									[9].arrDataOut[59]	:=	<0, 8, 8>TIIB(104)^API^Data^io^Outputs^Request Data[29];
									[9].arrDataOut[60]	:=	<0, 8, 0>TIIB(104)^API^Data^io^Outputs^Request Data[30];
									[9].arrDataOut[61]	:=	<0, 8, 8>TIIB(104)^API^Data^io^Outputs^Request Data[30];
									[9].arrDataOut[62]	:=	<0, 8, 0>TIIB(104)^API^Data^io^Outputs^Request Data[31];
									[9].arrDataOut[63]	:=	<0, 8, 8>TIIB(104)^API^Data^io^Outputs^Request Data[31];
									[9].PnIoBoxState 	:=	<0, 16, 0>TIIB(104)^Inputs^PnIoBoxState;
									[10].arrDataIn[0]	:=	<0, 8, 0>TIIB(105)^API^Data^io^Inputs^Response Data[0];
									[10].arrDataIn[1]	:=	<0, 8, 8>TIIB(105)^API^Data^io^Inputs^Response Data[0];
									[10].arrDataIn[2]	:=	<0, 8, 0>TIIB(105)^API^Data^io^Inputs^Response Data[1];
									[10].arrDataIn[3]	:=	<0, 8, 8>TIIB(105)^API^Data^io^Inputs^Response Data[1];
									[10].arrDataIn[4]	:=	<0, 8, 0>TIIB(105)^API^Data^io^Inputs^Response Data[2];
									[10].arrDataIn[5]	:=	<0, 8, 8>TIIB(105)^API^Data^io^Inputs^Response Data[2];
									[10].arrDataIn[6]	:=	<0, 8, 0>TIIB(105)^API^Data^io^Inputs^Response Data[3];
									[10].arrDataIn[7]	:=	<0, 8, 8>TIIB(105)^API^Data^io^Inputs^Response Data[3];
									[10].arrDataIn[8]	:=	<0, 8, 0>TIIB(105)^API^Data^io^Inputs^Response Data[4];
									[10].arrDataIn[9]	:=	<0, 8, 8>TIIB(105)^API^Data^io^Inputs^Response Data[4];
									[10].arrDataIn[10]	:=	<0, 8, 0>TIIB(105)^API^Data^io^Inputs^Response Data[5];
									[10].arrDataIn[11]	:=	<0, 8, 8>TIIB(105)^API^Data^io^Inputs^Response Data[5];
									[10].arrDataIn[12]	:=	<0, 8, 0>TIIB(105)^API^Data^io^Inputs^Response Data[6];
									[10].arrDataIn[13]	:=	<0, 8, 8>TIIB(105)^API^Data^io^Inputs^Response Data[6];
									[10].arrDataIn[14]	:=	<0, 8, 0>TIIB(105)^API^Data^io^Inputs^Response Data[7];
									[10].arrDataIn[15]	:=	<0, 8, 8>TIIB(105)^API^Data^io^Inputs^Response Data[7];
									[10].arrDataIn[16]	:=	<0, 8, 0>TIIB(105)^API^Data^io^Inputs^Response Data[8];
									[10].arrDataIn[17]	:=	<0, 8, 8>TIIB(105)^API^Data^io^Inputs^Response Data[8];
									[10].arrDataIn[18]	:=	<0, 8, 0>TIIB(105)^API^Data^io^Inputs^Response Data[9];
									[10].arrDataIn[19]	:=	<0, 8, 8>TIIB(105)^API^Data^io^Inputs^Response Data[9];
									[10].arrDataIn[20]	:=	<0, 8, 0>TIIB(105)^API^Data^io^Inputs^Response Data[10];
									[10].arrDataIn[21]	:=	<0, 8, 8>TIIB(105)^API^Data^io^Inputs^Response Data[10];
									[10].arrDataIn[22]	:=	<0, 8, 0>TIIB(105)^API^Data^io^Inputs^Response Data[11];
									[10].arrDataIn[23]	:=	<0, 8, 8>TIIB(105)^API^Data^io^Inputs^Response Data[11];
									[10].arrDataIn[24]	:=	<0, 8, 0>TIIB(105)^API^Data^io^Inputs^Response Data[12];
									[10].arrDataIn[25]	:=	<0, 8, 8>TIIB(105)^API^Data^io^Inputs^Response Data[12];
									[10].arrDataIn[26]	:=	<0, 8, 0>TIIB(105)^API^Data^io^Inputs^Response Data[13];
									[10].arrDataIn[27]	:=	<0, 8, 8>TIIB(105)^API^Data^io^Inputs^Response Data[13];
									[10].arrDataIn[28]	:=	<0, 8, 0>TIIB(105)^API^Data^io^Inputs^Response Data[14];
									[10].arrDataIn[29]	:=	<0, 8, 8>TIIB(105)^API^Data^io^Inputs^Response Data[14];
									[10].arrDataIn[30]	:=	<0, 8, 0>TIIB(105)^API^Data^io^Inputs^Response Data[15];
									[10].arrDataIn[31]	:=	<0, 8, 8>TIIB(105)^API^Data^io^Inputs^Response Data[15];
									[10].arrDataIn[32]	:=	<0, 8, 0>TIIB(105)^API^Data^io^Inputs^Response Data[16];
									[10].arrDataIn[33]	:=	<0, 8, 8>TIIB(105)^API^Data^io^Inputs^Response Data[16];
									[10].arrDataIn[34]	:=	<0, 8, 0>TIIB(105)^API^Data^io^Inputs^Response Data[17];
									[10].arrDataIn[35]	:=	<0, 8, 8>TIIB(105)^API^Data^io^Inputs^Response Data[17];
									[10].arrDataIn[36]	:=	<0, 8, 0>TIIB(105)^API^Data^io^Inputs^Response Data[18];
									[10].arrDataIn[37]	:=	<0, 8, 8>TIIB(105)^API^Data^io^Inputs^Response Data[18];
									[10].arrDataIn[38]	:=	<0, 8, 0>TIIB(105)^API^Data^io^Inputs^Response Data[19];
									[10].arrDataIn[39]	:=	<0, 8, 8>TIIB(105)^API^Data^io^Inputs^Response Data[19];
									[10].arrDataIn[40]	:=	<0, 8, 0>TIIB(105)^API^Data^io^Inputs^Response Data[20];
									[10].arrDataIn[41]	:=	<0, 8, 8>TIIB(105)^API^Data^io^Inputs^Response Data[20];
									[10].arrDataIn[42]	:=	<0, 8, 0>TIIB(105)^API^Data^io^Inputs^Response Data[21];
									[10].arrDataIn[43]	:=	<0, 8, 8>TIIB(105)^API^Data^io^Inputs^Response Data[21];
									[10].arrDataIn[44]	:=	<0, 8, 0>TIIB(105)^API^Data^io^Inputs^Response Data[22];
									[10].arrDataIn[45]	:=	<0, 8, 8>TIIB(105)^API^Data^io^Inputs^Response Data[22];
									[10].arrDataIn[46]	:=	<0, 8, 0>TIIB(105)^API^Data^io^Inputs^Response Data[23];
									[10].arrDataIn[47]	:=	<0, 8, 8>TIIB(105)^API^Data^io^Inputs^Response Data[23];
									[10].arrDataIn[48]	:=	<0, 8, 0>TIIB(105)^API^Data^io^Inputs^Response Data[24];
									[10].arrDataIn[49]	:=	<0, 8, 8>TIIB(105)^API^Data^io^Inputs^Response Data[24];
									[10].arrDataIn[50]	:=	<0, 8, 0>TIIB(105)^API^Data^io^Inputs^Response Data[25];
									[10].arrDataIn[51]	:=	<0, 8, 8>TIIB(105)^API^Data^io^Inputs^Response Data[25];
									[10].arrDataIn[52]	:=	<0, 8, 0>TIIB(105)^API^Data^io^Inputs^Response Data[26];
									[10].arrDataIn[53]	:=	<0, 8, 8>TIIB(105)^API^Data^io^Inputs^Response Data[26];
									[10].arrDataIn[54]	:=	<0, 8, 0>TIIB(105)^API^Data^io^Inputs^Response Data[27];
									[10].arrDataIn[55]	:=	<0, 8, 8>TIIB(105)^API^Data^io^Inputs^Response Data[27];
									[10].arrDataIn[56]	:=	<0, 8, 0>TIIB(105)^API^Data^io^Inputs^Response Data[28];
									[10].arrDataIn[57]	:=	<0, 8, 8>TIIB(105)^API^Data^io^Inputs^Response Data[28];
									[10].arrDataIn[58]	:=	<0, 8, 0>TIIB(105)^API^Data^io^Inputs^Response Data[29];
									[10].arrDataIn[59]	:=	<0, 8, 8>TIIB(105)^API^Data^io^Inputs^Response Data[29];
									[10].arrDataIn[60]	:=	<0, 8, 0>TIIB(105)^API^Data^io^Inputs^Response Data[30];
									[10].arrDataIn[61]	:=	<0, 8, 8>TIIB(105)^API^Data^io^Inputs^Response Data[30];
									[10].arrDataIn[62]	:=	<0, 8, 0>TIIB(105)^API^Data^io^Inputs^Response Data[31];
									[10].arrDataIn[63]	:=	<0, 8, 8>TIIB(105)^API^Data^io^Inputs^Response Data[31];
									[10].arrDataOut[0]	:=	<0, 8, 0>TIIB(105)^API^Data^io^Outputs^Request Data[0];
									[10].arrDataOut[1]	:=	<0, 8, 8>TIIB(105)^API^Data^io^Outputs^Request Data[0];
									[10].arrDataOut[2]	:=	<0, 8, 0>TIIB(105)^API^Data^io^Outputs^Request Data[1];
									[10].arrDataOut[3]	:=	<0, 8, 8>TIIB(105)^API^Data^io^Outputs^Request Data[1];
									[10].arrDataOut[4]	:=	<0, 8, 0>TIIB(105)^API^Data^io^Outputs^Request Data[2];
									[10].arrDataOut[5]	:=	<0, 8, 8>TIIB(105)^API^Data^io^Outputs^Request Data[2];
									[10].arrDataOut[6]	:=	<0, 8, 0>TIIB(105)^API^Data^io^Outputs^Request Data[3];
									[10].arrDataOut[7]	:=	<0, 8, 8>TIIB(105)^API^Data^io^Outputs^Request Data[3];
									[10].arrDataOut[8]	:=	<0, 8, 0>TIIB(105)^API^Data^io^Outputs^Request Data[4];
									[10].arrDataOut[9]	:=	<0, 8, 8>TIIB(105)^API^Data^io^Outputs^Request Data[4];
									[10].arrDataOut[10]	:=	<0, 8, 0>TIIB(105)^API^Data^io^Outputs^Request Data[5];
									[10].arrDataOut[11]	:=	<0, 8, 8>TIIB(105)^API^Data^io^Outputs^Request Data[5];
									[10].arrDataOut[12]	:=	<0, 8, 0>TIIB(105)^API^Data^io^Outputs^Request Data[6];
									[10].arrDataOut[13]	:=	<0, 8, 8>TIIB(105)^API^Data^io^Outputs^Request Data[6];
									[10].arrDataOut[14]	:=	<0, 8, 0>TIIB(105)^API^Data^io^Outputs^Request Data[7];
									[10].arrDataOut[15]	:=	<0, 8, 8>TIIB(105)^API^Data^io^Outputs^Request Data[7];
									[10].arrDataOut[16]	:=	<0, 8, 0>TIIB(105)^API^Data^io^Outputs^Request Data[8];
									[10].arrDataOut[17]	:=	<0, 8, 8>TIIB(105)^API^Data^io^Outputs^Request Data[8];
									[10].arrDataOut[18]	:=	<0, 8, 0>TIIB(105)^API^Data^io^Outputs^Request Data[9];
									[10].arrDataOut[19]	:=	<0, 8, 8>TIIB(105)^API^Data^io^Outputs^Request Data[9];
									[10].arrDataOut[20]	:=	<0, 8, 0>TIIB(105)^API^Data^io^Outputs^Request Data[10];
									[10].arrDataOut[21]	:=	<0, 8, 8>TIIB(105)^API^Data^io^Outputs^Request Data[10];
									[10].arrDataOut[22]	:=	<0, 8, 0>TIIB(105)^API^Data^io^Outputs^Request Data[11];
									[10].arrDataOut[23]	:=	<0, 8, 8>TIIB(105)^API^Data^io^Outputs^Request Data[11];
									[10].arrDataOut[24]	:=	<0, 8, 0>TIIB(105)^API^Data^io^Outputs^Request Data[12];
									[10].arrDataOut[25]	:=	<0, 8, 8>TIIB(105)^API^Data^io^Outputs^Request Data[12];
									[10].arrDataOut[26]	:=	<0, 8, 0>TIIB(105)^API^Data^io^Outputs^Request Data[13];
									[10].arrDataOut[27]	:=	<0, 8, 8>TIIB(105)^API^Data^io^Outputs^Request Data[13];
									[10].arrDataOut[28]	:=	<0, 8, 0>TIIB(105)^API^Data^io^Outputs^Request Data[14];
									[10].arrDataOut[29]	:=	<0, 8, 8>TIIB(105)^API^Data^io^Outputs^Request Data[14];
									[10].arrDataOut[30]	:=	<0, 8, 0>TIIB(105)^API^Data^io^Outputs^Request Data[15];
									[10].arrDataOut[31]	:=	<0, 8, 8>TIIB(105)^API^Data^io^Outputs^Request Data[15];
									[10].arrDataOut[32]	:=	<0, 8, 0>TIIB(105)^API^Data^io^Outputs^Request Data[16];
									[10].arrDataOut[33]	:=	<0, 8, 8>TIIB(105)^API^Data^io^Outputs^Request Data[16];
									[10].arrDataOut[34]	:=	<0, 8, 0>TIIB(105)^API^Data^io^Outputs^Request Data[17];
									[10].arrDataOut[35]	:=	<0, 8, 8>TIIB(105)^API^Data^io^Outputs^Request Data[17];
									[10].arrDataOut[36]	:=	<0, 8, 0>TIIB(105)^API^Data^io^Outputs^Request Data[18];
									[10].arrDataOut[37]	:=	<0, 8, 8>TIIB(105)^API^Data^io^Outputs^Request Data[18];
									[10].arrDataOut[38]	:=	<0, 8, 0>TIIB(105)^API^Data^io^Outputs^Request Data[19];
									[10].arrDataOut[39]	:=	<0, 8, 8>TIIB(105)^API^Data^io^Outputs^Request Data[19];
									[10].arrDataOut[40]	:=	<0, 8, 0>TIIB(105)^API^Data^io^Outputs^Request Data[20];
									[10].arrDataOut[41]	:=	<0, 8, 8>TIIB(105)^API^Data^io^Outputs^Request Data[20];
									[10].arrDataOut[42]	:=	<0, 8, 0>TIIB(105)^API^Data^io^Outputs^Request Data[21];
									[10].arrDataOut[43]	:=	<0, 8, 8>TIIB(105)^API^Data^io^Outputs^Request Data[21];
									[10].arrDataOut[44]	:=	<0, 8, 0>TIIB(105)^API^Data^io^Outputs^Request Data[22];
									[10].arrDataOut[45]	:=	<0, 8, 8>TIIB(105)^API^Data^io^Outputs^Request Data[22];
									[10].arrDataOut[46]	:=	<0, 8, 0>TIIB(105)^API^Data^io^Outputs^Request Data[23];
									[10].arrDataOut[47]	:=	<0, 8, 8>TIIB(105)^API^Data^io^Outputs^Request Data[23];
									[10].arrDataOut[48]	:=	<0, 8, 0>TIIB(105)^API^Data^io^Outputs^Request Data[24];
									[10].arrDataOut[49]	:=	<0, 8, 8>TIIB(105)^API^Data^io^Outputs^Request Data[24];
									[10].arrDataOut[50]	:=	<0, 8, 0>TIIB(105)^API^Data^io^Outputs^Request Data[25];
									[10].arrDataOut[51]	:=	<0, 8, 8>TIIB(105)^API^Data^io^Outputs^Request Data[25];
									[10].arrDataOut[52]	:=	<0, 8, 0>TIIB(105)^API^Data^io^Outputs^Request Data[26];
									[10].arrDataOut[53]	:=	<0, 8, 8>TIIB(105)^API^Data^io^Outputs^Request Data[26];
									[10].arrDataOut[54]	:=	<0, 8, 0>TIIB(105)^API^Data^io^Outputs^Request Data[27];
									[10].arrDataOut[55]	:=	<0, 8, 8>TIIB(105)^API^Data^io^Outputs^Request Data[27];
									[10].arrDataOut[56]	:=	<0, 8, 0>TIIB(105)^API^Data^io^Outputs^Request Data[28];
									[10].arrDataOut[57]	:=	<0, 8, 8>TIIB(105)^API^Data^io^Outputs^Request Data[28];
									[10].arrDataOut[58]	:=	<0, 8, 0>TIIB(105)^API^Data^io^Outputs^Request Data[29];
									[10].arrDataOut[59]	:=	<0, 8, 8>TIIB(105)^API^Data^io^Outputs^Request Data[29];
									[10].arrDataOut[60]	:=	<0, 8, 0>TIIB(105)^API^Data^io^Outputs^Request Data[30];
									[10].arrDataOut[61]	:=	<0, 8, 8>TIIB(105)^API^Data^io^Outputs^Request Data[30];
									[10].arrDataOut[62]	:=	<0, 8, 0>TIIB(105)^API^Data^io^Outputs^Request Data[31];
									[10].arrDataOut[63]	:=	<0, 8, 8>TIIB(105)^API^Data^io^Outputs^Request Data[31];
									[10].PnIoBoxState 	:=	<0, 16, 0>TIIB(105)^Inputs^PnIoBoxState;	'}
	fbRFID_Readers				:ARRAY[1..10] OF FB_ID200;
END_VAR

// ---- GVLs/GVL_Safety.TcGVL
VAR_GLOBAL
(*-----=== Common ===-----*)
(***************************************************Test**********************************************************)	
	q_bSafetyOverrideCnc1			AT %Q*	:BOOL;	// Enable
	q_bSafetyOverrideCnc2			AT %Q*	:BOOL;	// Enable
	q_bSafetyOverrideCnc3			AT %Q*	:BOOL;	// Enable
(**************************************************Inputs*********************************************************)	


(**************************************************Outputs********************************************************)
	q_bSafetyRun					AT %Q*	:BOOL;	// Safety run
	q_bBlink						AT %Q*	:BOOL;

(*-----=== CNC4 - CNC5 ===-----*)
(**************************************************Inputs*********************************************************)
	i_bLO1_CNC45					AT %I*	:BOOL;	
	i_bLO2_CNC45					AT %I*	:BOOL;	
	i_bLO1EDMErr_CNC45				AT %I*	:BOOL;	
	i_bLO2EDMErr_CNC45				AT %I*	:BOOL;	
	i_bSafetyGroupComErr_CNC45		AT %I*	:BOOL;
	i_bSafetyGroupFBErr_CNC45		AT %I*	:BOOL;	
	i_bSafetyGroupOtherErr_CNC45	AT %I*	:BOOL;
	i_bWaitClose_CNC45				AT %I*	:BOOL;
	bSafetyError_CNC45						:BOOL;	// Safety error
(**************************************************Outputs********************************************************)
	q_bSafetyMasterOn_CNC45			AT %Q*	:BOOL;	// Master on
	q_bCellEmptyAck_CNC45			AT %Q*	:BOOL;	// Cell empty ack
	q_bSafetyErrorAck_CNC45			AT %Q*	:BOOL;	// Safety ack


(*-----=== Main ===-----*)
(**************************************************Inputs*********************************************************)	
	i_bLO1_Main						AT %I*	:BOOL;	
	i_bLO2_Main						AT %I*	:BOOL;	
	i_bLO1EDMErr_Main				AT %I*	:BOOL;	
	i_bLO2EDMErr_Main				AT %I*	:BOOL;	
	i_bSafetyGroupComErr_Main		AT %I*	:BOOL;
	i_bSafetyGroupFBErr_Main		AT %I*	:BOOL;	
	i_bSafetyGroupOtherErr_Main		AT %I*	:BOOL;
	i_bWaitClose_Main				AT %I*	:BOOL;
	bSafetyError_Main						:BOOL;	// Safety error
(**************************************************Outputs********************************************************)
	q_bSafetyMasterOn_Main			AT %Q*	:BOOL;	// Master on
	q_bCellEmptyAck_Main			AT %Q*	:BOOL;	// Cell empty ack
	q_bSafetyErrorAck_Main			AT %Q*	:BOOL;	// Safety ack

(*-----=== CNC1 ===-----*)
(**************************************************Inputs*********************************************************)
	i_bLO1_CNC1						AT %I*	:BOOL;
	i_bRobotDoorOpened_CNC1			AT %I*	:BOOL;

(*-----=== CNC2 ===-----*)
(**************************************************Inputs*********************************************************)
	i_bLO1_CNC2						AT %I*	:BOOL;
	i_bRobotDoorOpened_CNC2			AT %I*	:BOOL;

(*-----=== CNC2 ===-----*)
(**************************************************Inputs*********************************************************)
	i_bLO1_CNC3						AT %I*	:BOOL;
	i_bRobotDoorOpened_CNC3			AT %I*	:BOOL;
END_VAR

// ---- POUs/MAIN.TcPOU
PROGRAM MAIN
VAR
	rtStep						:R_Trig;
	
	rtAck						:R_Trig;
	i							:UDINT;
	fbWakeUpTmr					:TON;	
	sTime						:STRING(8);
	bAckLED						:BOOL;
	darius						:UDINT;	
	
	// Alarm	
	aErrorActive				:ARRAY[1..nNbrOfAlarms] OF WORD;
	aErrorID1					:ARRAY[1..nNbrOfAlarms] OF STRING(255);
	aErrorID2					:ARRAY[1..nNbrOfAlarms] OF STRING(255);
	afbAlarms					:ARRAY[1..nNbrOfAlarms] OF FB_TcAlarm;
	fbSource					:FB_TcSourceInfo;

	(*Vise station components*)
	rtStepViseStation			:R_Trig;

END_VAR

//InitTCPIP();
Init();
Blink();
SafetyPRG();
Alarm();
BusDiag();
Door();
Light();
Mode();
ViseProgram();
RobotCncProgram();
Robot7AxisProgram();
RobotKardexProgram();
CNC_1();
CNC_2();
CNC_3();
ConveyorSystem();
UploadingProgram();
Mapping();

Test();
SQL_Test();


fbTime(bEnable := TRUE, dwCycle := 1);
dtSystemTime := SYSTEMTIME_TO_DT(TIMESTR:= fbTime.systemTime);
sTime := MID((SYSTEMTIME_TO_STRING(fbTime.systemTime)),8,12);

ACTION Alarm:
// Creating error acknowladge impulse
rtAck(CLK:= i_bVisePos1ErrorAckBtn OR i_bVisePos2ErrorAckBtn OR bAckHMI OR i_bErrorAckBtn_Main, Q=> bAckP);
IF rtAck.Q THEN
	afbAlarms[1].Confirm(0); afbAlarms[2].Confirm(0); afbAlarms[3].Confirm(0); afbAlarms[4].Confirm(0);
	afbAlarms[5].Confirm(0); afbAlarms[6].Confirm(0); afbAlarms[7].Confirm(0); 
	bAckHMI := FALSE;
END_IF

IF wError <> 0 OR bSafetyError_CNC45 OR ViseProgram.nState >= 200000 THEN
	bGlobalError := TRUE;
ELSE
	bGlobalError := FALSE;
END_IF

(* 
	wError.0 : Air pressure error
	wError.1 : Ethercat error
	wError.2 : 
	wError.3 : 
	wError.4 : 
	wError.5 : 
	wError.6 : 
	wError.7 : 
	wError.8 : 
	wError.9 : 
*)

aErrorActive[1].0 := wError.0;
aErrorActive[2].0 := wError.1;
aErrorActive[3].0 := i_bSafetyGroupComErr_CNC45;
aErrorActive[4].0 := i_bSafetyGroupFBErr_CNC45;
aErrorActive[5].0 := i_bSafetyGroupOtherErr_CNC45;
aErrorActive[6].0 := i_bLO1EDMErr_CNC45;
aErrorActive[7].0 := i_bLO2EDMErr_CNC45;

FOR i := 1 TO nNbrOfAlarms DO
	IF aErrorActive[i].0 THEN
		IF (afbAlarms[i].eConfirmationState <> 2 AND afbAlarms[i].nTimeCleared <> 0 AND afbAlarms[i].nTimeConfirmed <> 0) OR //Ha már volt alarm, akkor van bennük érték
			(afbAlarms[i].eConfirmationState = 1 AND afbAlarms[i].nTimeCleared = 0 AND afbAlarms[i].nTimeConfirmed = 0)	//Első futás esetén
		THEN
			IF aErrorActive[i].1 AND aErrorActive[i].2 THEN
				afbAlarms[i].ipArguments.Clear().AddString(aErrorID1[i]).AddString(aErrorID2[i]);
			ELSIF aErrorActive[i].1 THEN
				afbAlarms[i].ipArguments.Clear().AddString(aErrorID1[i]);
			ELSE
				afbAlarms[i].ipArguments.Clear();
			END_IF
			afbAlarms[i].Raise(0);
		END_IF	
	ELSE
		IF (afbAlarms[i].eConfirmationState = 2 OR afbAlarms[i].eConfirmationState = 3) AND afbAlarms[i].nTimeCleared = 0 THEN
			afbAlarms[i].Clear(0, FALSE);
		END_IF		
	END_IF
END_FOR
END_ACTION

ACTION BusDiag:
fbWakeUpTmr(IN:= NOT bFirstCycle, PT:= T#60S, Q=> , ET=> );
// eCAT network error
IF fbWakeUpTmr.Q AND (i_nBusState <> 8) THEN
	wError.1 := TRUE;	
END_IF
END_ACTION

ACTION Door:
fbDoor(
	bDoorButton:= i_bDoorRequest, 
	bOpenEnable:= TRUE (*and robot.....*),
	bEmergencyOk:= i_bLO1_CNC45,
	bWaitClose:= i_bWaitClose_CNC45,
	bDoorsClosed:= i_bDoorClosed, 
	bDoorsLocked:= i_bLO2_CNC45, 
	bBlink_1:= bBL100p100,
	bBlink_2:= bBL500p500, 
	bCloseOut=> q_bDoorLock, 
	bDoorButtonLED=> q_bDoorRequestLED,
	bCellAckLED => q_bCellAckLED, 
	bObenRequestOut=> bDoorOpenReq);
END_ACTION

ACTION Init:
IF bFirstCycle THEN
	afbAlarms[1].CreateEx(TC_Events.MyEvents.AirPE, TRUE, 0);
	afbAlarms[2].CreateEx(TC_Events.MyEvents.GenEtherCATErr, TRUE, 0);
	afbAlarms[3].CreateEx(TC_Events.MyEvents.SafetyGroupComErr, TRUE, 0);
	afbAlarms[4].CreateEx(TC_Events.MyEvents.SafetyGroupFbErr, TRUE, 0);
	afbAlarms[5].CreateEx(TC_Events.MyEvents.SafetyGroupOtherErr, TRUE, 0);
	afbAlarms[6].CreateEx(TC_Events.MyEvents.LO1EDMErr, TRUE, 0);
	afbAlarms[7].CreateEx(TC_Events.MyEvents.LO2EDMErr, TRUE, 0);
	
	fb3DCam.p_ConnectTimeout := T#2S;
	fb3DCam.p_SendTimeout := T#2S;
	fb3DCam.p_ReceiveTimeout := T#20S;
	fb3DCam.p_CloseTimeout := T#2S;
	fb3DCam.p_Name := '3D Camera';
	fb3DCam.p_RemoteHost := '192.168.81.19';
	fb3DCam.p_RemotePort := 24056;

	bFirstCycle := FALSE;
END_IF
END_ACTION

ACTION Light:
//Master on light
q_bMasterOnLED := (i_bLO1_CNC45 (*AND i_bLO2*)) OR (bBL500p500 AND 
					NOT i_bEmyStop1 AND NOT i_bEmyStop2 AND NOT i_bEmyStop3 AND
					NOT i_bEmyStop4 AND NOT i_bEmyStop5 AND NOT i_bEmyStop6);

//Error acknowledge light
bAckLED := (bGlobalError AND bBL500p500) OR 
			i_bEmyStop1 OR i_bEmyStop2 OR i_bEmyStop3 OR
			i_bEmyStop4 OR i_bEmyStop5 OR i_bEmyStop6;

q_bVise1ErrorAckLED := q_bVise2ErrorAckBtnLED := bAckLED;
	
fbNotSmartLight(
	bEmyStop:= i_bEmyStop1 OR i_bEmyStop2 OR i_bEmyStop3 OR i_bEmyStop4 OR i_bEmyStop5 OR i_bEmyStop6,
	bEmyOK:= i_bLO1_CNC45 AND i_bLO2_CNC45, 
	bError:= bGlobalError, 
	bOutOfStock:= ,
	bBuzzer := FALSE,
	bBlink := bBL500p500);
END_ACTION

ACTION Mapping:
;
END_ACTION

ACTION Mode:
// Switching mode
IF bManualModeRequest THEN
	IF (Robot7AxisProgram.nState = 0 OR Robot7AxisProgram.nState = 10000 OR Robot7AxisProgram.nState = 150000 OR Robot7AxisProgram.nState >= 200000) 
	THEN
		nMode := 2;
		bManualMode := TRUE;
		bGlobalEHA := FALSE;
	ELSE
		nMode := 1;
	END_IF
ELSE
	nMode := 0;
	bManualMode := FALSE;
	bGlobalEHA := TRUE;
END_IF

// Switching mode Vise
IF bManualModeRequestVise THEN
	IF (ViseProgram.nState = 0 OR ViseProgram.nState = 10000 OR ViseProgram.nState = 150000 OR ViseProgram.nState >= 200000) 
	THEN
		nModeVise := 2;
		bManualModeVise := TRUE;
		//bGlobalEHAVise := FALSE;
	ELSE
		nModeVise := 1;
	END_IF
ELSE
	nModeVise := 0;
	bManualModeVise := FALSE;
	//bGlobalEHAVise := TRUE;
END_IF


// Step mode for testing
rtStep(CLK:= bStepHMI OR i_bMasterOn_CNC45 OR i_bMasterOn_Main, Q=> bStepP);
IF bStepMode AND bStepP OR NOT bStepMode THEN
	bStepEnable := TRUE;
ELSE
	bStepEnable := FALSE;
END_IF

// Step mode for testing in Vise Station
rtStepViseStation(CLK:= bStepHMIViseStation OR i_bMasterOn_CNC45 OR i_bMasterOn_Main, Q=> bStepPViseStation);
IF bStepModeViseStation AND bStepPViseStation OR (NOT bStepModeViseStation) THEN
	bStepEnableViseStation := TRUE;
ELSE
	bStepEnableViseStation := FALSE;
END_IF
END_ACTION

END_PROGRAM

// ---- POUs/Blink.TcPOU
PROGRAM Blink
VAR
	tBL1					:FB_GenPulse; (*50ms/50ms*)
	tBL2					:FB_GenPulse; (*100ms/100ms*)
	tBL3					:FB_GenPulse; (*250ms/250ms*)
	tBL4					:FB_GenPulse; (*500ms/500ms*)
	tBL5					:FB_GenPulse; (*1000ms/1000ms*)
	tBL6					:FB_GenPulse; (*750ms/250ms*)
	tBL7					:FB_GenPulse; (*750ms/250ms*)
	tBL8					:FB_GenPulse; (*1000ms/1000ms*)
	rtBL1,rtBL2,rtBL3,rtBL4	:R_TRIG;
END_VAR


tBL1(ENQ:= TRUE, PTH:= T#50MS, PTL:= T#50MS, Q=> bBL50p50);
tBL2(ENQ:= TRUE, PTH:= T#100MS, PTL:= T#100MS, Q=> bBL100p100);
tBL3(ENQ:= TRUE, PTH:= T#250MS, PTL:= T#250MS, Q=> bBL250p250);
tBL4(ENQ:= TRUE, PTH:= T#500MS, PTL:= T#500MS, Q=> bBL500p500);
tBL5(ENQ:= TRUE, PTH:= T#1000MS, PTL:= T#1000MS, Q=> bBL1000p1000);
tBL6(ENQ:= TRUE, PTH:= T#250MS, PTL:= T#750MS, Q=> bBL250p750);
tBL7(ENQ:= TRUE, PTH:= T#750MS, PTL:= T#250MS, Q=> bBL750p250);
tBL8(ENQ:= TRUE, PTH:= T#2000MS, PTL:= T#2000MS, Q=> bBL2000p2000);
rtBL1(CLK:= GVL_Main.bBL50p50, Q=> bTakt100ms);
rtBL2(CLK:= GVL_Main.bBL100p100, Q=> bTakt200ms);
rtBL3(CLK:= GVL_Main.bBL250p250, Q=> bTakt500ms);
rtBL4(CLK:= GVL_Main.bBL500p500, Q=> bTakt1s);

IF bTakt100ms THEN
	wLifeSignal:=wLifeSignal + 1;      
END_IF
IF wLifeSignal>100 THEN
	wLifeSignal:=0;
END_IF

END_PROGRAM

// ---- POUs/FBs/Utilities/FB_GenPulse.TcPOU
FUNCTION_BLOCK FB_GenPulse
VAR_INPUT
	ENQ : BOOL := TRUE;
	PTH : TIME;
	PTL : TIME;
END_VAR
VAR_OUTPUT
	Q : BOOL;	
END_VAR
VAR
	timON: TON;
	timOFF: TON;
	init: BOOL;
END_VAR

IF NOT(Init) THEN
	timOFF.IN:=FALSE;
	timON.IN:=FALSE;
	Init:=TRUE;
END_IF;
timON(IN:= enq AND NOT(timOFF.Q), PT:=PTH);
timOFF(IN:= timON.Q, PT:=PTL);
Q:=timON.Q AND NOT(timOFF.Q);

END_FUNCTION_BLOCK

// ---- POUs/SafetyPRG.TcPOU
PROGRAM SafetyPRG
VAR
	fbAirTimer						:TON;
END_VAR

// Safety GroupPort run condition
q_bSafetyRun := TRUE;
q_bCellEmptyAck_CNC45 := i_bCellAck;
q_bSafetyMasterOn_CNC45 := i_bMasterOn_CNC45 AND bBL100p100;
q_bSafetyMasterOn_Main := i_bMasterOn_Main AND bBL100p100;
q_bBlink := bBL500p500;


(*Safety Override for CNC 1 to 3 Doors*)
GVL_Safety.q_bSafetyOverrideCnc1 := TRUE;
GVL_Safety.q_bSafetyOverrideCnc2 := TRUE;
GVL_Safety.q_bSafetyOverrideCnc3 := TRUE;

// Safety Error
bSafetyError_CNC45 := i_bSafetyGroupComErr_CNC45 OR i_bSafetyGroupFBErr_CNC45 OR i_bSafetyGroupOtherErr_CNC45 OR 
				i_bLO1EDMErr_CNC45 OR i_bLO2EDMErr_CNC45;

bSafetyError_Main := i_bSafetyGroupComErr_Main OR i_bSafetyGroupFBErr_Main OR i_bSafetyGroupOtherErr_Main OR 
				i_bLO1EDMErr_Main OR i_bLO2EDMErr_Main;

q_bSafetyErrorAck_CNC45 := bSafetyError_CNC45 AND bBL100p100 OR i_bVisePos1ErrorAckBtn OR i_bVisePos2ErrorAckBtn;				

q_bSafetyErrorAck_Main := bSafetyError_Main AND bBL100p100 OR i_bErrorAckBtn_Main;				

(*Air pressure error*)
fbAirTimer(IN:= i_bLO1_CNC45, PT:= T#10S);
IF i_bLO1_CNC45 THEN
	IF fbAirTimer.Q AND NOT i_bAirPressureOk THEN
		wError.0 := TRUE;
	END_IF
END_IF

IF bAckP THEN
	wError := 0;
END_IF

END_PROGRAM

// ---- POUs/RobotViseStation/ViseProgram.TcPOU
PROGRAM ViseProgram
VAR CONSTANT
	nStartIndex					:USINT := 1;
	nMaxIndex					:USINT := 14;
END_VAR
VAR	(* Control *)
	nState						:UDINT;
	nStatePrevious				:UDINT;
	sState						:STRING(500);
	fbCycleTime					:TON;
	nCycleTime					:REAL;
	eCommand					:E_Vise_Command;
	index						:UINT := 1;
	nCounter					:UINT;
	
	tWaitStabTime				:TON;
	tVisePushTime				:TON;
	tFillUpTime					:TON;
	bFirstCycle					:BOOL := TRUE;
END_VAR
VAR
	fbUnloadTrig				: R_TRIG;
END_VAR
VAR (* RGB *)
	arrColors					:ARRAY [1..24] OF ST_RGB_Light;
	nRgbCounter					:UINT;
	aViseErrorIndex				:ARRAY[1..14] OF BOOL;
END_VAR
VAR //LastStates
	anLastStates				:ARRAY[0..500] OF UDINT;
    iLastStates					:INT;
END_VAR
VAR // MySQL
	fbUpdateVise			: FB_SP_spUpdateVise;
	stParameterValues		: ST_ParaVal_UpdateVise;
	fbGetNextVise			: FB_SP_spGetNextVise;
END_VAR

Pneu();
RGB();
MySQL();

(*Init*)
IF bFirstCycle THEN
	eCommand := E_Vise_Command.Load;
	bFirstCycle := FALSE;
END_IF

(*Error handling*)
IF nState > 0 AND nState < 150000 THEN
	nStatePrevious := nState;
	FOR nCounter := nStartIndex TO nMaxIndex BY 1 DO
		IF fbViseStation[nCounter].bError THEN
			nState := 200000;
			aViseErrorIndex[nCounter] := TRUE;
		ELSE
			aViseErrorIndex[nCounter] := FALSE;
		END_IF
	END_FOR
END_IF

(*Maintance*)
IF bManualModeVise THEN
	nState := 150000;
END_IF

(*Emergency*)
IF NOT i_bLO1_CNC45 OR NOT i_bLO2_CNC45 THEN
	nState := 0;
END_IF

(*Last states*)
IF(nState >= 1000) AND (nState < 150000) THEN
(*Steps before any state*)
	IF anLastStates[0] <> nState THEN
		FOR iLastStates:=500 TO 1 BY -1 DO
			anLastStates[iLastStates]:= anLastStates[iLastStates-1];
		END_FOR
		anLastStates[0]:= nState;
	END_IF
END_IF	

//(*Base timeout*) 
//tWaitStabTime(IN:= nState = 40 OR nState = 80, PT:= T#1S, Q=> , ET=> );
//IF tWaitStabTime.Q THEN
//	nState := 200000;
//END_IF

(*Push out time*) 
tVisePushTime(IN:= (nState = 20060) OR (nState = 50060), PT:= T#400MS, Q=> , ET=> );

(*Fill up time*) 
tFillUpTime(IN:= (nState = 80) OR (nState = 140), PT:= T#2S, Q=> , ET=> );




aViseStatus[1].eState := E_Vise_State.OutOfService;

CASE nState OF
	(* Emergency circuit broken - Base state *)
	0:(* Operation stop - Emergency circuit check *)
		sState := CONCAT(UDINT_TO_STRING(nState) ,' - Vészkör bontva');
		FOR index := nStartIndex TO nMaxIndex BY 1 DO
			fbViseStation[index].StopperInner.bWorkPosCmd := FALSE;
			fbViseStation[index].StopperOuter.bWorkPosCmd := FALSE;
			fbViseStation[index].Vise.bBasePosCmd := FALSE;
			fbViseStation[index].Vise.bWorkPosCmd := FALSE;
		END_FOR
		IF i_bLO1_CNC45 AND i_bLO2_CNC45 AND NOT bManualModeVise THEN
			nState := nState + 20;
		END_IF
		
	20:
		sState := CONCAT(UDINT_TO_STRING(nState) ,' - Alaphelyzet felvétel - Satu betolva - Stopperek');
		FOR index := nStartIndex TO nMaxIndex BY 1 DO
			IF fbViseStation[index].stViseStationSensors.bInPos THEN
				IF (aViseStatus[index].eState <> E_Vise_State.OutOfService) THEN
					fbViseStation[index].StopperInner.bWorkPosCmd := TRUE;
				END_IF
			ELSE
				nState := 200000;
				EXIT;
			END_IF
		END_FOR
		IF index = (nMaxIndex + 1) THEN
			nState := nState + 20;
		END_IF
		
	40:	
		sState := CONCAT(UDINT_TO_STRING(nState) ,' - Alaphelyzet felvétel - Satu betolva - Stopperek');
		FOR index := nStartIndex TO nMaxIndex BY 1 DO
			IF (aViseStatus[index].eState <> E_Vise_State.OutOfService) THEN
				IF NOT fbViseStation[index].stViseStationSensors.bStopper_In_Hold THEN
					EXIT;
				END_IF
			END_IF
		END_FOR
		IF index = (nMaxIndex + 1) THEN
			nState := nState + 20;
		END_IF
		
	60:	
		sState := CONCAT(UDINT_TO_STRING(nState) ,' - Alaphelyzet felvétel - Satu betolva - Satu hengereinek feltöltése ');
		FOR index := 1 TO 7 BY 1 DO
			IF (aViseStatus[index].eState <> E_Vise_State.OutOfService) THEN
				fbViseStation[index].Vise.bWorkPosCmd := TRUE;
				fbViseStation[index].Vise.bBasePosCmd := TRUE;
			END_IF
		END_FOR
		
		nState := nState + 20;
		
	80:
		IF tFillUpTime.Q THEN
			nState := nState + 20;
		END_IF
	
	100:	
		sState := CONCAT(UDINT_TO_STRING(nState) ,' - Alaphelyzet felvétel - Satu betolva - Satu hengerek alaphelyzetbe');
		FOR index := 1 TO 7 BY 1 DO
			IF (aViseStatus[index].eState <> E_Vise_State.OutOfService) THEN
				fbViseStation[index].Vise.bWorkPosCmd := FALSE;
				fbViseStation[index].Vise.bBasePosCmd := TRUE;
			END_IF
		END_FOR
		
		nState := nState + 10;
		
	110:
		sState := CONCAT(UDINT_TO_STRING(nState) ,' - Satu alaphelyzetek ellenőrzése');
		
		FOR index := 1 TO 7 BY 1 DO
			IF (aViseStatus[index].eState <> E_Vise_State.OutOfService) THEN
				IF fbViseStation[index].Vise.bBasePosStab THEN
					nState := 120;
				ELSE
					EXIT;
				END_IF		
			END_IF
		END_FOR
		
	120:	
		sState := CONCAT(UDINT_TO_STRING(nState) ,' - Alaphelyzet felvétel - Satu betolva - Satu hengereinek feltöltése ');
		FOR index := 8 TO 14 BY 1 DO
			IF (aViseStatus[index].eState <> E_Vise_State.OutOfService) THEN
				fbViseStation[index].Vise.bWorkPosCmd := TRUE;
				fbViseStation[index].Vise.bBasePosCmd := TRUE;
			END_IF
		END_FOR
		nState := nState + 20;
		
	140:
		IF tFillUpTime.Q THEN
			nState := nState + 20;
		END_IF
	
	160:	
		sState := CONCAT(UDINT_TO_STRING(nState) ,' - Alaphelyzet felvétel - Satu betolva - Satu hengerek alaphelyzetbe');
		FOR index := 8 TO 14 BY 1 DO
			IF (aViseStatus[index].eState <> E_Vise_State.OutOfService) THEN
				fbViseStation[index].Vise.bWorkPosCmd := FALSE;
				fbViseStation[index].Vise.bBasePosCmd := TRUE;
			END_IF
		END_FOR
		
		nState := nState + 10;
		
	170:
		sState := CONCAT(UDINT_TO_STRING(nState) ,' - Satu alaphelyzetek ellenőrzése');
		
		FOR index := 8 TO 14 BY 1 DO
			IF (aViseStatus[index].eState <> E_Vise_State.OutOfService) THEN
				IF fbViseStation[index].Vise.bBasePosStab THEN
					nState := 180;
				ELSE
					EXIT;
				END_IF		
			END_IF
		END_FOR
		
	180:	
		FOR index := nStartIndex TO nMaxIndex BY 1 DO
			IF (aViseStatus[index].eState <> E_Vise_State.OutOfService) THEN
				IF NOT fbViseStation[index].fbVise.bBasePosStab THEN
					EXIT;
				END_IF
			END_IF
		END_FOR
		IF index = (nMaxIndex + 1) THEN
			nState := nState + 20;
		END_IF
		
	200:
		nState := 10000;
		
	(* Automatic mode - Base position *)
	10000:
		IF eCommand = E_Vise_Command.UnLoad THEN
			nState := 50000;
		ELSIF eCommand = E_Vise_Command.Load THEN
			nState := 20000;
		ELSIF eCommand = E_Vise_Command.InProcess THEN
			nState := 30000;
		END_IF

	(*-----=== Feltöltés ===-----*)
{region "Feltöltés"}
	20000: (*Load*)
		FOR index := nStartIndex TO nMaxIndex BY 1 DO
			IF (aViseStatus[index].eState = E_Vise_State.Empty OR aViseStatus[index].eState = E_Vise_State.OutForLoad) AND (aViseStatus[index].eState <> E_Vise_State.OutOfService) THEN
				nState := nState + 20;
				EXIT;
			END_IF
		END_FOR
		IF index = (nMaxIndex + 1) THEN
			eCommand := E_Vise_Command.InProcess;
			nState := 10000;
		END_IF
			
	20020: (*Stopper in release*)
		sState := CONCAT(UDINT_TO_STRING(nState) ,' - Belső stopper elengedése');
		fbViseStation[index].StopperInner.bWorkPosCmd := FALSE;
		nState := nState + 20;
		
	20040: (*Push out vise*)
		sState := CONCAT(UDINT_TO_STRING(nState) ,' - Belső stopper elengedése');
		IF fbViseStation[index].stViseStationSensors.bStopper_In_Release THEN
			IF index < 8 THEN
				q_bViseOut_1_7 := TRUE;
			ELSIF index > 7 THEN
				q_bViseOut_8_14 := TRUE;
			END_IF
			nState := nState + 20;
		END_IF
		
	20060:	
		sState := CONCAT(UDINT_TO_STRING(nState) ,' - Satu kilökése');
		IF tVisePushTime.Q THEN
			nState := nState + 20;
		END_IF
		
	20080: (*Waiting for out sensor*)
		q_bViseOut_1_7 := FALSE;
		q_bViseOut_8_14 := FALSE;
		sState := CONCAT(UDINT_TO_STRING(nState) ,' - Húzd ki a satut');
		aViseStatus[index].eState := E_Vise_State.OutForLoad;
		
		IF fbViseStation[index].stViseStationSensors.bOutPos THEN
			fbViseStation[index].StopperOuter.bWorkPosCmd := TRUE;
			nState := nState + 20;
		END_IF
		
	20100: (*Stopper out hold*)
		IF fbViseStation[index].fbStopper_Out.bWorkPosStab THEN
			nState := nState + 20;
		END_IF
		
	20120: (*Waiting for operator*)
		sState := CONCAT(UDINT_TO_STRING(nState) ,' - Satu feltöltése - Ha kész nyomd meg a gombot');
		IF (index > 7 AND i_bVisePos2InBtn) OR (index < 8 AND i_bVisePos1InBtn) THEN
			fbViseStation[index].StopperOuter.bWorkPosCmd := FALSE;
			nState := nState + 20;
		END_IF	
		
	20140: (*Stopper out release*)
		sState := CONCAT(UDINT_TO_STRING(nState) ,' - Satu elengedve - Told be a satut');
		IF fbViseStation[index].stViseStationSensors.bStopper_Out_Release THEN
			nState := nState + 20;
		END_IF
		
	20160: (*Waiting for operator to push vise in*)
		sState := CONCAT(UDINT_TO_STRING(nState) ,' - Told be a satut');
		IF fbViseStation[index].stViseStationSensors.bInPos THEN
			fbViseStation[index].StopperInner.bWorkPosCmd := TRUE;
			nState := nState + 20;
		END_IF
		
	20180:
		IF fbViseStation[index].fbStopper_In.bWorkPosStab THEN
			aViseStatus[index].eState := E_Vise_State.ReadyToCnc;
			eCommand := E_Vise_Command.UnLoad;
			nState := 10000;
		END_IF		
{endregion}

	(*-----=== InProcess ===-----*)
{region "Gyártás"}
	30000: (*In process*)
		FOR index := nStartIndex TO nMaxIndex BY 1 DO
			IF (aViseStatus[index].eState = E_Vise_State.Empty OR aViseStatus[index].eState = E_Vise_State.OutForLoad) AND (aViseStatus[index].eState <> E_Vise_State.OutOfService) THEN
				nState := nState + 20;
				EXIT;
			END_IF
		END_FOR
		IF index = (nMaxIndex + 1) THEN
			eCommand := E_Vise_Command.UnLoad;
			nState := 10000;
		END_IF

{endregion}

	(*-----=== Kiürítés ===-----*)
{region "Kiürítés"}		
	50000: (*Unload*)
		FOR index := nStartIndex TO nMaxIndex BY 1 DO
			IF (aViseStatus[index].eState = E_Vise_State.WaitingForUnLoad OR aViseStatus[index].eState = E_Vise_State.OutForUnload) AND (aViseStatus[index].eState <> E_Vise_State.OutOfService) THEN
				nState := nState + 20;
				EXIT;
			END_IF
		END_FOR
		// Unload is done, next cycle starts
		IF index = (nMaxIndex + 1) THEN			
			eCommand := E_Vise_Command.Load;
			nState := 10000;
		END_IF	
		
	50020: (*Stopper in release*)
		sState := CONCAT(UDINT_TO_STRING(nState) ,' - Belső stopper elengedése');
		fbViseStation[index].StopperInner.bWorkPosCmd := FALSE;
		nState := nState + 20;
		
	50040: (*Push out vise*)
		sState := CONCAT(UDINT_TO_STRING(nState) ,' - Belső stopper elengedése');
		IF fbViseStation[index].stViseStationSensors.bStopper_In_Release THEN
			IF index < 8 THEN
				q_bViseOut_1_7 := TRUE;
			ELSIF index > 7 THEN
				q_bViseOut_8_14 := TRUE;
			END_IF
			nState := nState + 20;
		END_IF
		
	50060:	
		sState := CONCAT(UDINT_TO_STRING(nState) ,' - Satu kilökése');
		IF tVisePushTime.Q THEN
			nState := nState + 20;
		END_IF
		
	50080: (*Waiting for out sensor*)
		q_bViseOut_1_7 := FALSE;
		q_bViseOut_8_14 := FALSE;
		sState := CONCAT(UDINT_TO_STRING(nState) ,' - Húzd ki a satut');
		aViseStatus[index].eState := E_Vise_State.OutForUnload;
		
		IF fbViseStation[index].stViseStationSensors.bOutPos THEN
			fbViseStation[index].StopperOuter.bWorkPosCmd := TRUE;
			nState := nState + 20;
		END_IF
		
	50100: (*Stopper out hold*)
		IF fbViseStation[index].fbStopper_Out.bWorkPosStab THEN
			nState := nState + 20;
		END_IF
		
	50120: (*Waiting for operator*)
		sState := CONCAT(UDINT_TO_STRING(nState) ,' - Satu kiürítése - Ha kész nyomd meg a gombot');
		IF (index > 7 AND i_bVisePos2InBtn) OR (index < 8 AND i_bVisePos1InBtn) THEN
			fbViseStation[index].StopperOuter.bWorkPosCmd := FALSE;
			nState := nState + 20;
		END_IF	
		
	50140: (*Stopper out release*)
		sState := CONCAT(UDINT_TO_STRING(nState) ,' - Satu elengedve - Told be a satut');
		IF fbViseStation[index].stViseStationSensors.bStopper_Out_Release THEN
			nState := nState + 20;
		END_IF
		
	50160: (*Waiting for operator to push vise in*)
		sState := CONCAT(UDINT_TO_STRING(nState) ,' - Told be a satut');
		IF fbViseStation[index].stViseStationSensors.bInPos THEN
			fbViseStation[index].StopperInner.bWorkPosCmd := TRUE;
			nState := nState + 20;
		END_IF
		
	50180:
		IF fbViseStation[index].fbStopper_In.bWorkPosStab THEN
			aViseStatus[index].eState := E_Vise_State.Empty;
			eCommand := E_Vise_Command.Load;
			nState := 10000;
		END_IF	
{endregion}

	
	150000: (* Maintenance *)
		sState := CONCAT(UDINT_TO_STRING(nState) ,' - Maintenance');
		IF NOT bManualModeVise THEN
			nState := 0;
		END_IF
		
	200000:(* Error handling *)
		sState := CONCAT(UDINT_TO_STRING(nState) ,CONCAT(' - Error, from this state: ' , sState));
		nState := 200020;

	200020:(* Error handling *)
		IF bAckP THEN
			CASE nStatePrevious OF
				0..9999: nState := 0;
				10000..60000: nState := 10000;
			ELSE nState := 0;
			END_CASE
		END_IF	
		
	ELSE //Not a real step, for test purposes
		sState := CONCAT(UDINT_TO_STRING(nState) ,' - Not a real step, for test purposes');
END_CASE

(*Timers***************************************************)
fbCycleTime(IN:= nState > 10000 AND nState <= 95000, PT:= T#1D, Q=> , ET=> );
IF nState > 10000 AND nState <= 95000 THEN
	nCycleTime := TIME_TO_REAL(fbCycleTime.ET)/1000;
END_IF

ACTION MySQL:
fbGetNextVise(
	Target:= , 
	nRecordStartIndex:= , 
	tTimeout:= , 
	bExecute:= , 
	bBusy=> , 
	bError=> , 
	ipResult=> , 
	nViseNr=> );

fbUpdateVise(
	nRecordStartIndex:= , 
	tTimeout:= , 
	bExecute:= , 
	bBusy=> , 
	bError=> , 
	ipResult=> , 
	stParameterValues:= stParameterValues);
END_ACTION

ACTION Pneu:
(**************************************************Vise station*********************************************************)	
fbViseStation[1](
	sName:= 'Vise 1', 
	bEn:= i_bLO1_CNC45 AND NOT (aViseStatus[1].eState = E_Vise_State.OutOfService), 
	bEHA:= bGlobalEHAVise, 
	bManualMode:= bManualModeVise, 
	bAck:= bAckP, 
	sSourceName:= 'Vise 1-7', 
	stViseBasePosEvent:= TC_Events.MyEvents.Satu1BasePosErr, 
	stViseWorkPosEvent:= TC_Events.MyEvents.Satu1WorkPosErr, 
	stStopperInWorkPosEvent:= TC_Events.MyEvents.Satu1_Stopper_In_WorkPosErr, 
	stStopperOutWorkPosEvent:= TC_Events.MyEvents.Satu1_Stopper_Out_WorkPosErr,
	stViseStationSensors:= i_stViseStationSensors_1);
	
fbViseStation[2](
	sName:= 'Vise 2', 
	bEn:= i_bLO1_CNC45 AND NOT (aViseStatus[2].eState = E_Vise_State.OutOfService), 
	bEHA:= bGlobalEHAVise, 
	bManualMode:= bManualModeVise, 
	bAck:= bAckP, 
	sSourceName:= 'Vise 1-7', 
	stViseBasePosEvent:= TC_Events.MyEvents.Satu2BasePosErr, 
	stViseWorkPosEvent:= TC_Events.MyEvents.Satu2WorkPosErr, 
	stStopperInWorkPosEvent:= TC_Events.MyEvents.Satu2_Stopper_In_WorkPosErr, 
	stStopperOutWorkPosEvent:= TC_Events.MyEvents.Satu2_Stopper_Out_WorkPosErr,
	stViseStationSensors:= i_stViseStationSensors_2);
	
fbViseStation[3](
	sName:= 'Vise 3', 
	bEn:= i_bLO1_CNC45 AND NOT (aViseStatus[3].eState = E_Vise_State.OutOfService), 
	bEHA:= bGlobalEHAVise, 
	bManualMode:= bManualModeVise, 
	bAck:= bAckP, 
	sSourceName:= 'Vise 1-7', 
	stViseBasePosEvent:= TC_Events.MyEvents.Satu3BasePosErr, 
	stViseWorkPosEvent:= TC_Events.MyEvents.Satu3WorkPosErr, 
	stStopperInWorkPosEvent:= TC_Events.MyEvents.Satu3_Stopper_In_WorkPosErr, 
	stStopperOutWorkPosEvent:= TC_Events.MyEvents.Satu3_Stopper_Out_WorkPosErr,
	stViseStationSensors:= i_stViseStationSensors_3);
	
fbViseStation[4](
	sName:= 'Vise 4', 
	bEn:= i_bLO1_CNC45 AND NOT (aViseStatus[4].eState = E_Vise_State.OutOfService), 
	bEHA:= bGlobalEHAVise, 
	bManualMode:= bManualModeVise, 
	bAck:= bAckP, 
	sSourceName:= 'Vise 1-7', 
	stViseBasePosEvent:= TC_Events.MyEvents.Satu4BasePosErr, 
	stViseWorkPosEvent:= TC_Events.MyEvents.Satu4WorkPosErr, 
	stStopperInWorkPosEvent:= TC_Events.MyEvents.Satu4_Stopper_In_WorkPosErr, 
	stStopperOutWorkPosEvent:= TC_Events.MyEvents.Satu4_Stopper_Out_WorkPosErr,
	stViseStationSensors:= i_stViseStationSensors_4);
	
fbViseStation[5](
	sName:= 'Vise 5', 
	bEn:= i_bLO1_CNC45 AND NOT (aViseStatus[5].eState = E_Vise_State.OutOfService), 
	bEHA:= bGlobalEHAVise, 
	bManualMode:= bManualModeVise, 
	bAck:= bAckP, 
	sSourceName:= 'Vise 1-7', 
	stViseBasePosEvent:= TC_Events.MyEvents.Satu5BasePosErr, 
	stViseWorkPosEvent:= TC_Events.MyEvents.Satu5WorkPosErr, 
	stStopperInWorkPosEvent:= TC_Events.MyEvents.Satu5_Stopper_In_WorkPosErr, 
	stStopperOutWorkPosEvent:= TC_Events.MyEvents.Satu5_Stopper_Out_WorkPosErr,
	stViseStationSensors:= i_stViseStationSensors_5);
	
fbViseStation[6](
	sName:= 'Vise 6', 
	bEn:= i_bLO1_CNC45 AND NOT (aViseStatus[6].eState = E_Vise_State.OutOfService), 
	bEHA:= bGlobalEHAVise, 
	bManualMode:= bManualModeVise, 
	bAck:= bAckP, 
	sSourceName:= 'Vise 1-7', 
	stViseBasePosEvent:= TC_Events.MyEvents.Satu6BasePosErr, 
	stViseWorkPosEvent:= TC_Events.MyEvents.Satu6WorkPosErr, 
	stStopperInWorkPosEvent:= TC_Events.MyEvents.Satu6_Stopper_In_WorkPosErr, 
	stStopperOutWorkPosEvent:= TC_Events.MyEvents.Satu6_Stopper_Out_WorkPosErr,
	stViseStationSensors:= i_stViseStationSensors_6);
	
fbViseStation[7](
	sName:= 'Vise 7', 
	bEn:= i_bLO1_CNC45 AND NOT (aViseStatus[7].eState = E_Vise_State.OutOfService), 
	bEHA:= bGlobalEHAVise, 
	bManualMode:= bManualModeVise, 
	bAck:= bAckP, 
	sSourceName:= 'Vise 1-7', 
	stViseBasePosEvent:= TC_Events.MyEvents.Satu7BasePosErr, 
	stViseWorkPosEvent:= TC_Events.MyEvents.Satu7WorkPosErr, 
	stStopperInWorkPosEvent:= TC_Events.MyEvents.Satu7_Stopper_In_WorkPosErr, 
	stStopperOutWorkPosEvent:= TC_Events.MyEvents.Satu7_Stopper_Out_WorkPosErr,
	stViseStationSensors:= i_stViseStationSensors_7);
	
fbViseStation[8](
	sName:= 'Vise 8', 
	bEn:= i_bLO1_CNC45 AND NOT (aViseStatus[8].eState = E_Vise_State.OutOfService), 
	bEHA:= bGlobalEHAVise, 
	bManualMode:= bManualModeVise, 
	bAck:= bAckP, 
	sSourceName:= 'Vise 8-14', 
	stViseBasePosEvent:= TC_Events.MyEvents.Satu8BasePosErr, 
	stViseWorkPosEvent:= TC_Events.MyEvents.Satu8WorkPosErr, 
	stStopperInWorkPosEvent:= TC_Events.MyEvents.Satu8_Stopper_In_WorkPosErr, 
	stStopperOutWorkPosEvent:= TC_Events.MyEvents.Satu8_Stopper_Out_WorkPosErr,
	stViseStationSensors:= i_stViseStationSensors_8);
	
fbViseStation[9](
	sName:= 'Vise 9', 
	bEn:= i_bLO1_CNC45 AND NOT (aViseStatus[9].eState = E_Vise_State.OutOfService), 
	bEHA:= bGlobalEHAVise, 
	bManualMode:= bManualModeVise, 
	bAck:= bAckP, 
	sSourceName:= 'Vise 8-14', 
	stViseBasePosEvent:= TC_Events.MyEvents.Satu9BasePosErr, 
	stViseWorkPosEvent:= TC_Events.MyEvents.Satu9WorkPosErr, 
	stStopperInWorkPosEvent:= TC_Events.MyEvents.Satu9_Stopper_In_WorkPosErr, 
	stStopperOutWorkPosEvent:= TC_Events.MyEvents.Satu9_Stopper_Out_WorkPosErr,
	stViseStationSensors:= i_stViseStationSensors_9);
	
fbViseStation[10](
	sName:= 'Vise 10', 
	bEn:= i_bLO1_CNC45 AND NOT (aViseStatus[10].eState = E_Vise_State.OutOfService), 
	bEHA:= bGlobalEHAVise, 
	bManualMode:= bManualModeVise, 
	bAck:= bAckP, 
	sSourceName:= 'Vise 8-14', 
	stViseBasePosEvent:= TC_Events.MyEvents.Satu10BasePosErr, 
	stViseWorkPosEvent:= TC_Events.MyEvents.Satu10WorkPosErr, 
	stStopperInWorkPosEvent:= TC_Events.MyEvents.Satu10_Stopper_In_WorkPosErr, 
	stStopperOutWorkPosEvent:= TC_Events.MyEvents.Satu10_Stopper_Out_WorkPosErr,
	stViseStationSensors:= i_stViseStationSensors_10);
	
fbViseStation[11](
	sName:= 'Vise 11', 
	bEn:= i_bLO1_CNC45 AND NOT (aViseStatus[11].eState = E_Vise_State.OutOfService), 
	bEHA:= bGlobalEHAVise, 
	bManualMode:= bManualModeVise, 
	bAck:= bAckP, 
	sSourceName:= 'Vise 8-14', 
	stViseBasePosEvent:= TC_Events.MyEvents.Satu11BasePosErr, 
	stViseWorkPosEvent:= TC_Events.MyEvents.Satu11WorkPosErr, 
	stStopperInWorkPosEvent:= TC_Events.MyEvents.Satu11_Stopper_In_WorkPosErr, 
	stStopperOutWorkPosEvent:= TC_Events.MyEvents.Satu11_Stopper_Out_WorkPosErr,
	stViseStationSensors:= i_stViseStationSensors_11);
	
fbViseStation[12](
	sName:= 'Vise 12', 
	bEn:= i_bLO1_CNC45 AND NOT (aViseStatus[12].eState = E_Vise_State.OutOfService), 
	bEHA:= bGlobalEHAVise, 
	bManualMode:= bManualModeVise, 
	bAck:= bAckP, 
	sSourceName:= 'Vise 8-14', 
	stViseBasePosEvent:= TC_Events.MyEvents.Satu12BasePosErr, 
	stViseWorkPosEvent:= TC_Events.MyEvents.Satu12WorkPosErr, 
	stStopperInWorkPosEvent:= TC_Events.MyEvents.Satu12_Stopper_In_WorkPosErr, 
	stStopperOutWorkPosEvent:= TC_Events.MyEvents.Satu12_Stopper_Out_WorkPosErr,
	stViseStationSensors:= i_stViseStationSensors_12);
	
fbViseStation[13](
	sName:= 'Vise 13', 
	bEn:= i_bLO1_CNC45 AND NOT (aViseStatus[13].eState = E_Vise_State.OutOfService), 
	bEHA:= bGlobalEHAVise, 
	bManualMode:= bManualModeVise, 
	bAck:= bAckP, 
	sSourceName:= 'Vise 8-14', 
	stViseBasePosEvent:= TC_Events.MyEvents.Satu13BasePosErr, 
	stViseWorkPosEvent:= TC_Events.MyEvents.Satu13WorkPosErr, 
	stStopperInWorkPosEvent:= TC_Events.MyEvents.Satu13_Stopper_In_WorkPosErr, 
	stStopperOutWorkPosEvent:= TC_Events.MyEvents.Satu13_Stopper_Out_WorkPosErr,
	stViseStationSensors:= i_stViseStationSensors_13);
	
fbViseStation[14](
	sName:= 'Vise 14', 
	bEn:= i_bLO1_CNC45 AND NOT (aViseStatus[14].eState = E_Vise_State.OutOfService), 
	bEHA:= bGlobalEHAVise, 
	bManualMode:= bManualModeVise, 
	bAck:= bAckP, 
	sSourceName:= 'Vise 8-14', 
	stViseBasePosEvent:= TC_Events.MyEvents.Satu14BasePosErr, 
	stViseWorkPosEvent:= TC_Events.MyEvents.Satu14WorkPosErr, 
	stStopperInWorkPosEvent:= TC_Events.MyEvents.Satu14_Stopper_In_WorkPosErr, 
	stStopperOutWorkPosEvent:= TC_Events.MyEvents.Satu14_Stopper_Out_WorkPosErr,
	stViseStationSensors:= i_stViseStationSensors_14);
END_ACTION

ACTION RGB:
FOR nRgbCounter := nStartIndex TO nMaxIndex BY 1 DO
	CASE aViseStatus[nRgbCounter].eState OF
		// Violet - Violet - Violet
	 	E_Vise_State.OutOfService:
			arrColors[nRgbCounter].nColor1 := cViolet;
			arrColors[nRgbCounter].nColor1State := TRUE;
			arrColors[nRgbCounter].nColor2 := cViolet;
			arrColors[nRgbCounter].nColor2State := TRUE;
			arrColors[nRgbCounter].nColor3 := cViolet;
			arrColors[nRgbCounter].nColor3State := TRUE;
			
		// Fail : Red - None - Red; Pass: Green - None - Green
		E_Vise_State.WaitingForUnLoad:
			IF aViseStatus[index].bFail THEN
				arrColors[nRgbCounter].nColor1 := cRed;
				arrColors[nRgbCounter].nColor1State := TRUE;
				arrColors[nRgbCounter].nColor2 := cRed;
				arrColors[nRgbCounter].nColor2State := FALSE;
				arrColors[nRgbCounter].nColor3 := cRed;
				arrColors[nRgbCounter].nColor3State := TRUE;	
			ELSIF aViseStatus[index].bPass THEN
				arrColors[nRgbCounter].nColor1 := cGreen;
				arrColors[nRgbCounter].nColor1State := TRUE;
				arrColors[nRgbCounter].nColor2 := cGreen;
				arrColors[nRgbCounter].nColor2State := FALSE;
				arrColors[nRgbCounter].nColor3 := cGreen;
				arrColors[nRgbCounter].nColor3State := TRUE; 
			END_IF
			
		// Dark blue - Indigo blink - Dark blue
		E_Vise_State.OutForLoad:
			arrColors[nRgbCounter].nColor1 := cDarkBlue;
			arrColors[nRgbCounter].nColor1State := TRUE;
			arrColors[nRgbCounter].nColor2 := cIndigo;
			arrColors[nRgbCounter].nColor2State := bBL1000p1000;
			arrColors[nRgbCounter].nColor3 := cDarkBlue;
			arrColors[nRgbCounter].nColor3State := TRUE;
		
		// Fail : Red - Blink red - Red; Pass: Green - Blink green - Green	
		E_Vise_State.OutForUnload:
			IF aViseStatus[index].bFail THEN
				arrColors[nRgbCounter].nColor1 := cRed;
				arrColors[nRgbCounter].nColor1State := TRUE;
				arrColors[nRgbCounter].nColor2 := cRed;
				arrColors[nRgbCounter].nColor2State := bBL1000p1000;
				arrColors[nRgbCounter].nColor3 := cRed;
				arrColors[nRgbCounter].nColor3State := TRUE;	
			ELSIF aViseStatus[index].bPass THEN
				arrColors[nRgbCounter].nColor1 := cGreen;
				arrColors[nRgbCounter].nColor1State := TRUE;
				arrColors[nRgbCounter].nColor2 := cGreen;
				arrColors[nRgbCounter].nColor2State := bBL1000p1000;
				arrColors[nRgbCounter].nColor3 := cGreen;
				arrColors[nRgbCounter].nColor3State := TRUE; 
			END_IF
			
		// White - White - White
		E_Vise_State.Empty: 
			arrColors[nRgbCounter].nColor1 := cWhite;
			arrColors[nRgbCounter].nColor1State := TRUE;
			arrColors[nRgbCounter].nColor2 := cWhite;
			arrColors[nRgbCounter].nColor2State := TRUE;
			arrColors[nRgbCounter].nColor3 := cWhite;
			arrColors[nRgbCounter].nColor3State := TRUE;
			
		// Dark blue - Dark blue - Dark blue
		E_Vise_State.InCnc:
			arrColors[nRgbCounter].nColor1 := cDarkBlue;
			arrColors[nRgbCounter].nColor1State := TRUE;
			arrColors[nRgbCounter].nColor2 := cDarkBlue;
			arrColors[nRgbCounter].nColor2State := TRUE;
			arrColors[nRgbCounter].nColor3 := cDarkBlue;
			arrColors[nRgbCounter].nColor3State := TRUE;
			
		// Dark blue - Dark blue - Dark blue
		E_Vise_State.ReadyToCnc:
			arrColors[nRgbCounter].nColor1 := cDarkBlue;
			arrColors[nRgbCounter].nColor1State := TRUE;
			arrColors[nRgbCounter].nColor2 := cDarkBlue;
			arrColors[nRgbCounter].nColor2State := TRUE;
			arrColors[nRgbCounter].nColor3 := cDarkBlue;
			arrColors[nRgbCounter].nColor3State := TRUE;
			
	END_CASE
	
	// Blink Red - Orange - Blink Red
	IF aViseErrorIndex[nRgbCounter] THEN 
		arrColors[nRgbCounter].nColor1 := cRed;
		arrColors[nRgbCounter].nColor1State := bBL1000p1000;
		arrColors[nRgbCounter].nColor2 := cOrange;
		arrColors[nRgbCounter].nColor2State := TRUE;
		arrColors[nRgbCounter].nColor3 := cRed;
		arrColors[nRgbCounter].nColor3State := bBL1000p1000;
	END_IF
	
	// No LO1 or LO2 Red - Red - Red
	IF NOT i_bLO1_CNC45 OR NOT i_bLO2_CNC45 THEN
		arrColors[nRgbCounter].nColor1 := cRed;
		arrColors[nRgbCounter].nColor1State := TRUE;
		arrColors[nRgbCounter].nColor2 := cRed;
		arrColors[nRgbCounter].nColor2State := TRUE;
		arrColors[nRgbCounter].nColor3 := cRed;
		arrColors[nRgbCounter].nColor3State := TRUE;
	END_IF
END_FOR
fbRgbLights(arrColors:= arrColors);
END_ACTION

END_PROGRAM

// ---- POUs/FBs/MySQL/UpdateVise/FB_SP_spUpdateVise.TcPOU
FUNCTION_BLOCK FB_SP_spUpdateVise
VAR_INPUT
	nRecordStartIndex			: UDINT;
	tTimeout					: TIME;
	bExecute					: BOOL;
END_VAR
VAR_OUTPUT
	bBusy						: BOOL;
	bError						: BOOL;
	ipResult					: I_TcMessage;
END_VAR
VAR_IN_OUT
	stParameterValues			: ST_ParaVal_UpdateVise;
END_VAR
VAR
	R_TRIG_Execute				: R_TRIG;
	nState						: INT;
	nErrState					: INT;
	fbSQLDatabase				: FB_SQLDatabaseEvt(sNetID := '', tTimeout := TIME#5s0ms);
	fbSQLStoredProcedure		: FB_SQLStoredProcedureEvt(sNetID := '', tTimeout := TIME#5s0ms);
	fbSQLResult					: FB_SQLResultEvt(sNetID := '', tTimeout := TIME#5s0ms);
	arrParaInfo					: ARRAY[0..5] OF ST_SQLSPParameter;
END_VAR

CASE nState OF
	0:
		R_TRIG_Execute(CLK:=bExecute);
		IF R_TRIG_Execute.Q THEN
			nState := 1;
			bBusy:=TRUE;
			bError:=FALSE;
			nErrState:=0;
		END_IF
	1:
		IF fbSQLDatabase.Connect(1) THEN
			ipResult:=fbSQLDatabase.ipTcResult;
			IF fbSQLDatabase.bError THEN
				nErrState:=1;
				nState:=255;
			ELSE
				arrParaInfo[0].sParameterName := 'ViseNumber';
				arrParaInfo[0].eParameterType := E_SPParameterType.Input;
				arrParaInfo[0].eParameterDataType := E_ColumnType.TinyInt;
				arrParaInfo[0].nParameterSize := 1;

				arrParaInfo[1].sParameterName := 'SerialNumber';
				arrParaInfo[1].eParameterType := E_SPParameterType.Input;
				arrParaInfo[1].eParameterDataType := E_ColumnType.NVarChar;
				arrParaInfo[1].nParameterSize := 256;

				arrParaInfo[2].sParameterName := 'DutIdentifier';
				arrParaInfo[2].eParameterType := E_SPParameterType.Input;
				arrParaInfo[2].eParameterDataType := E_ColumnType.BigInt;
				arrParaInfo[2].nParameterSize := 8;

				arrParaInfo[3].sParameterName := 'CamIdentifier';
				arrParaInfo[3].eParameterType := E_SPParameterType.Input;
				arrParaInfo[3].eParameterDataType := E_ColumnType.BigInt;
				arrParaInfo[3].nParameterSize := 8;

				arrParaInfo[4].sParameterName := 'CncNumber';
				arrParaInfo[4].eParameterType := E_SPParameterType.Input;
				arrParaInfo[4].eParameterDataType := E_ColumnType.TinyInt;
				arrParaInfo[4].nParameterSize := 1;
				
				nState:= 2;
			END_IF
		END_IF
	2:
		IF fbSQLDatabase.CreateSP('spUpdateVise', ADR(arrParaInfo), SIZEOF(arrParaInfo), ADR(fbSQLStoredProcedure)) THEN
			IF fbSQLDatabase.bError THEN
				nErrState:=2;
				nState:=255;
			ELSE
				nState:=3;
			END_IF
		END_IF
	3:
		IF fbSQLStoredProcedure.ExecuteDataReturn(ADR(stParameterValues), SIZEOF(stParameterValues), ADR(fbSQLResult))THEN
			ipResult:=fbSQLStoredProcedure.ipTcResult;
			IF fbSQLStoredProcedure.bError THEN
				nErrState:=3;
				nState:=255;
			ELSE
				nState:= 5;
			END_IF
		END_IF
	
	5:
		IF fbSQLStoredProcedure.Release() THEN
			IF fbSQLStoredProcedure.bError THEN
				nErrState:=5;
				nState:=255;
			ELSE
				nState:= 200;
			END_IF
		END_IF
	200:
		IF fbSQLDatabase.Disconnect() THEN
			nState := 0;
			bBusy:= FALSE;
		END_IF
	255:
		bError:= TRUE;
		bBusy:= FALSE;
		IF nErrState > 1 THEN
			nState:=200;
		ELSE
			nState:=0;
		END_IF
END_CASE

END_FUNCTION_BLOCK

// ---- POUs/FBs/MySQL/NextVise/FB_SP_spGetNextVise.TcPOU
FUNCTION_BLOCK FB_SP_spGetNextVise
VAR_INPUT
	Target						: BYTE;		// 0:empty;		1:wait operator;		4,5: wait cnc;
	nRecordStartIndex			: UDINT;
	tTimeout					: TIME;
	bExecute					: BOOL;
END_VAR
VAR_OUTPUT
	bBusy						: BOOL;
	bError						: BOOL;
	ipResult					: I_TcMessage;
	nViseNr						: BYTE;
END_VAR
VAR
	R_TRIG_Execute				: R_TRIG;
	nState						: INT;
	nErrState					: INT;
	fbSQLDatabase				: FB_SQLDatabaseEvt(sNetID := '', tTimeout := TIME#5s0ms);
	fbSQLStoredProcedure		: FB_SQLStoredProcedureEvt(sNetID := '', tTimeout := TIME#5s0ms);
	fbSQLResult					: FB_SQLResultEvt(sNetID := '', tTimeout := TIME#5s0ms);
	arrParaInfo					: ARRAY[0..1] OF ST_SQLSPParameter;
	stParameterValues			: ST_ParaVal_GetNextVise;
END_VAR

CASE nState OF
	0:
		R_TRIG_Execute(CLK:=bExecute);
		IF R_TRIG_Execute.Q THEN
			nState := 1;
			bBusy:=TRUE;
			bError:=FALSE;
			nErrState:=0;
		END_IF
	1:
		IF fbSQLDatabase.Connect(1) THEN
			ipResult:=fbSQLDatabase.ipTcResult;
			IF fbSQLDatabase.bError THEN
				nErrState:=1;
				nState:=255;
			ELSE
				arrParaInfo[0].sParameterName := 'Target';
				arrParaInfo[0].eParameterType := E_SPParameterType.Input;
				arrParaInfo[0].eParameterDataType := E_ColumnType.TinyInt;
				arrParaInfo[0].nParameterSize := 1;

				arrParaInfo[1].sParameterName := 'ViseNumber';
				arrParaInfo[1].eParameterType := E_SPParameterType.Output;
				arrParaInfo[1].eParameterDataType := E_ColumnType.TinyInt;
				arrParaInfo[1].nParameterSize := 1;
				nState:= 2;
			END_IF
		END_IF
	2:
		IF fbSQLDatabase.CreateSP('spGetNextVise', ADR(arrParaInfo), SIZEOF(arrParaInfo), ADR(fbSQLStoredProcedure)) THEN
			IF fbSQLDatabase.bError THEN
				nErrState:=2;
				nState:=255;
			ELSE
				nState:=3;
			END_IF
		END_IF
	3:
		stParameterValues.Target := Target;
		IF fbSQLStoredProcedure.ExecuteDataReturn(ADR(stParameterValues), SIZEOF(stParameterValues), ADR(fbSQLResult))THEN
			ipResult:=fbSQLStoredProcedure.ipTcResult;
			IF fbSQLStoredProcedure.bError THEN
				nErrState:=3;
				nState:=255;
			ELSE
				nState:= 4;
			END_IF
		END_IF
	4:
		IF fbSQLResult.Read(nRecordStartIndex, 1, ADR(nViseNr), SIZEOF(nViseNr), TRUE, TRUE) THEN
			ipResult:=fbSQLResult.ipTcResult;
			IF fbSQLResult.bError THEN
				nErrState:=4;
				nState:= 255;
			ELSE
				nState:= 5;
			END_IF
		END_IF
	5:
		IF fbSQLStoredProcedure.Release() THEN
			IF fbSQLStoredProcedure.bError THEN
				nErrState:=5;
				nState:=255;
			ELSE
				nState:= 200;
			END_IF
		END_IF
	200:
		IF fbSQLDatabase.Disconnect() THEN
			nState := 0;
			bBusy:= FALSE;
		END_IF
	255:
		bError:= TRUE;
		bBusy:= FALSE;
		IF nErrState > 1 THEN
			nState:=200;
		ELSE
			nState:=0;
		END_IF
END_CASE

END_FUNCTION_BLOCK

// ---- POUs/Test.TcPOU
PROGRAM Test
VAR
	fbExecuter	:	NT_StartProcess;
	bTrig		: BOOL;
END_VAR
VAR
	sImageTestPath	: T_MaxString := 'C:\Test\felfogasi_terv\M1 K.PNG';
END_VAR
VAR
	fbCommandLine	: FB_CommandLineExecuter;
	bCommandLineTrig : BOOL;
	bMoveFileTrig	: BOOL;
	sSourceFIle		: STRING := 'C:\Test\asd.png';
	sTargetFile		: STRING := 'C:\Test\testerino\asd.png';
END_VAR
VAR
	fbEnum			: FB_EnumFindFileEntry;
	sFilePath		: T_MaxString := 'C:\Test\testerino\asd.png';
    bFileCheckTrig 	: BOOL;
    nFileCheckState	: UDINT;
	bFileFound		: BOOL;
END_VAR
VAR
	fbViseMySqlSpTest		: FB_SQL;
	bDbInit					: BOOL := FALSE;
	sName					: STRING := 'SmartFactory';
	nDBID					: UINT := 1;
	tTimeout				: TIME := T#10s;
	bGetNextVase			: BOOL := FALSE;

	sProcedureName			: STRING := 'spGetNextVise';				//Store Procedure name
    aParaInfo				: ARRAY [0..1] OF ST_SQLSPParameter;		//Parameter Info Array
	nCncNumber				: BYTE;										//Parameter in
	nViseNumber				: BYTE;										//Parameter out
END_VAR
//VAR
//	nSqlState			: INT := 0;
//	aSpParaList			: ARRAY [0..1] OF ST_DBParameter;
//	fbSpNextVise		: FB_DBStoredProcedures;
//	bGetNextVase		: BOOL := FALSE;
//	bSqlError			: BOOL;
	
//	nCncNumber			: BYTE;										//Parameter in
//	nViseNumber			: BYTE;										//Parameter out
//END_VAR
var
	_test_usint : USINT;
	_test : bool;
	fbCmdExecute			: Tc2_Utilities.NT_StartProcess;
END_VAR

fbCmdExecute(
	NETID:= '', 
	PATHSTR:= 'C:\Users\Administrator\AppData\Local\Programs\Python\Python312\python.exe', 
	DIRNAME:= 'C:\Python_Test', 
	COMNDLINE:= 'cmd_test.py', 
	START:= , 
	TMOUT:= , 
	BUSY=> , 
	ERR=> , 
	ERRID=> );
_test_usint.0 := 1;
_test := _test_usint.0;
//CASE nSqlState OF
//	0:
//			IF bGetNextVase THEN
//				nSqlState := nSqlState + 20;
//			END_IF

//	20:	
//			SqlInitSpPara();
//			fbSpNextVise(bExecute:= FALSE);
//			IF bStepMode AND bStepP OR NOT bStepMode THEN
//				nSqlState := nSqlState + 20;
//			END_IF

//	40:
//			fbSpNextVise(bExecute:= TRUE);
//			IF NOT fbSpNextVise.bBusy THEN
//				fbSpNextVise(bExecute:= FALSE);
//				bGetNextVase := FALSE;
//				IF NOT fbSpNextVise.bError THEN
//					nSqlState := nSqlState + 20;
//				ELSE
//					bSqlError := TRUE;
//					nSqlState := 0;
//				END_IF
//			END_IF	
//END_CASE
//fbSpNextVise(
//	sNetID:= , 
//	hDBID:= 1, 
//	sProcedureName:= 'spGetNextVise', 
//	pParameterList:= ADR(aSpParaList), 
//	cbParameterList:= SIZEOF(aSpParaList), 
//	tTimeout:= T#5S);


fbViseMySqlSpTest();
IF NOT bDbInit THEN
	IF fbViseMySqlSpTest.Init(sName, nDBID, tTimeout) THEN
		bDbInit := TRUE;
	END_IF
END_IF

// Stored procedure parameters
aParaInfo[0].sParameterName     := 'CncNumber'; 
aParaInfo[0].eParameterType     := E_SPParameterType.Input;
aParaInfo[0].eParameterDataType := E_ColumnType.TinyInt;
aParaInfo[0].nParameterSize     := SIZEOF(nCncNumber);

aParaInfo[1].sParameterName     := 'ViseNumber'; 
aParaInfo[1].eParameterType     := E_SPParameterType.Input;
aParaInfo[1].eParameterDataType := E_ColumnType.TinyInt;
aParaInfo[1].nParameterSize     := SIZEOF(nCncNumber);

IF bGetNextVase THEN
	IF fbViseMySqlSpTest.StoredProcedure(sProcedureName,
										ADR(aParaInfo), SIZEOF(aParaInfo),
										ADR(nCncNumber), SIZEOF(nCncNumber),
										ADR(nViseNumber), SIZEOF(nViseNumber)) THEN
		bGetNextVase := FALSE;
	END_IF
END_IF

IF bTrig THEN
	fbExecuter(START := TRUE);
	fbExecuter(START := FALSE);
	bTrig := FALSE;
END_IF

fbExecuter(
	NETID:= '', 
	PATHSTR:= 'C:\Windows\System32\cmd.exe', 
	DIRNAME:= 'C:\Windows\System32',
	COMNDLINE:= '/C echo deez nuts && pause', 
	TMOUT:= T#10S, );
	
IF bCommandLineTrig AND_THEN fbCommandLine.ExecuteCommand('/C echo deez nuts && pause') = E_Executer_State.Done THEN
	bCommandLineTrig := FALSE;
END_IF

IF bMoveFileTrig THEN
	IF fbCommandLine.MoveFile(sSourceFIle , sTargetFile) = E_Executer_State.Done THEN
		bMoveFileTrig := FALSE;
	ELSIF fbCommandLine.MoveFile(sSourceFIle , sTargetFile) = E_Executer_State.Error THEN
		bMoveFileTrig := FALSE;
	END_IF
END_IF


CASE nFileCheckState OF 
	0:
		IF bFileCheckTrig THEN
			bFileFound := FALSE;
			bFileCheckTrig := FALSE;
			fbEnum.sPathName := sFilePath;
			fbEnum.eCmd := E_EnumCmdType.eEnumCmd_First;
			nFileCheckState := nFileCheckState + 20;		
		END_IF
		
	20:
		fbEnum( bExecute := FALSE );
        fbEnum( bExecute := TRUE );
		nFileCheckState := nFileCheckState + 20;	
		
	40:
		fbEnum( bExecute := FALSE );
        IF NOT fbEnum.bBusy THEN
            IF NOT fbEnum.bError THEN
                IF NOT fbEnum.bEOE THEN
                   	nFileCheckState	:= 0;
					bFileFound := TRUE;
                ELSE (* no more entries *)
                    ;
                END_IF
            ELSE (* log error *)
                ;
            END_IF
        END_IF
END_CASE

//IF i_bTest_Up OR i_bTest_Down THEN
//	q_bConveyor_1 := TRUE;
//END_IF
//IF i_bTest_Stop THEN
//	q_bConveyor_1 := FALSE;
//	q_bConveyor_2 := q_bConveyor_1;
//	q_bConveyor_3 := q_bConveyor_1;
//	q_bConveyor_4 := q_bConveyor_1;
//	q_bConveyor_5 := q_bConveyor_1;
//	q_bConveyor_6 := q_bConveyor_1;
//	q_bConveyor_7 := q_bConveyor_1;
//	q_bConveyor_8 := q_bConveyor_1;
//	q_bConveyor_9 := q_bConveyor_1;
//	q_bConveyor_10 := q_bConveyor_1;
//	q_bConveyor_11 := q_bConveyor_1;
//END_IF

//q_bConveyor_2 := q_bConveyor_1;
//q_bConveyor_3 := q_bConveyor_1;
//q_bConveyor_4 := q_bConveyor_1;
//q_bConveyor_5 := q_bConveyor_1;
//q_bConveyor_6 := q_bConveyor_1;
//q_bConveyor_7 := q_bConveyor_1;
//q_bConveyor_8 := q_bConveyor_1;
//q_bConveyor_9 := q_bConveyor_1;
//q_bConveyor_10 := q_bConveyor_1;
//q_bConveyor_11 := q_bConveyor_1;

ACTION SqlInitSpPara:
//aSpParaList[0].sParameterName    := 'CncNumber';
//aSpParaList[0].eParameterDataType:= Tc2_Database.eDBColumn_TinyInt;
//aSpParaList[0].eParameterType    := Tc2_Database.eDBParameter_Input;
//aSpParaList[0].cbParameterValue  := SIZEOF(nCncNumber);
//aSpParaList[0].pParameterValue   := ADR(nCncNumber);

//aSpParaList[1].sParameterName    := 'ViseNumber';
//aSpParaList[1].eParameterDataType:= Tc2_Database.eDBColumn_TinyInt;
//aSpParaList[1].eParameterType    := Tc2_Database.eDBParameter_Output;
//aSpParaList[1].cbParameterValue  := SIZEOF(nViseNumber);
//aSpParaList[1].pParameterValue   := ADR(nViseNumber);
END_ACTION

END_PROGRAM

// ---- POUs/FBs/Utilities/FB_CommandLineExecuter.TcPOU
FUNCTION_BLOCK FB_CommandLineExecuter
VAR
	_executer		: NT_StartProcess;
	_file_finder	: FB_EnumFindFileEntry;
END_VAR
VAR
	_move_file_state : UINT;
END_VAR

METHOD PUBLIC ExecuteCommand : E_Executer_State
VAR_INPUT
	CommandLine		: T_MaxString;
END_VAR
ExecuteCommand := E_Executer_State.Busy;

_executer(
	NETID:= '',
	START := TRUE, 
	PATHSTR:= 'C:\Windows\System32\cmd.exe', 
	DIRNAME:= 'C:\Windows\System32',
	COMNDLINE:= CommandLine, 
	TMOUT:= T#10S);
	
IF NOT _executer.BUSY THEN
	_executer(START := FALSE);
	ExecuteCommand := E_Executer_State.Done;
END_IF

IF _executer.ERR THEN
	_executer(START := FALSE);
	ExecuteCommand := E_Executer_State.Error;
END_IF
END_METHOD

METHOD PUBLIC MoveFile : E_Executer_State
VAR_INPUT
	Source 		: T_MaxString;
	Destination : T_MaxString;
END_VAR
VAR
	_command	: T_MaxString;
END_VAR
// Build Command String
_command := '/C ';                  // Special command indicating command string input
_command := CONCAT(_command, 'move ');      // Add move command
_command := CONCAT(_command, Source);  // Add target file
_command := CONCAT(_command, ' ');          // Required space for command 
_command := CONCAT(_command, Destination); // Add target location
CASE _move_file_state OF
	0: 
		_move_file_state := _move_file_state + 20;
	
	20:
		IF THIS^.ExecuteCommand(_command) = E_Executer_State.Done THEN
			_move_file_state := _move_file_state + 20;
		END_IF	
	
	40:
		_file_finder.sPathName := Destination;
		_file_finder.eCmd := E_EnumCmdType.eEnumCmd_First;
		_move_file_state := _move_file_state + 20;
		
	60:
        _file_finder( bExecute := TRUE );
		_move_file_state := _move_file_state + 20;	
		
	80:
		_file_finder( bExecute := FALSE );
        IF NOT _file_finder.bBusy THEN
            IF NOT _file_finder.bError AND NOT _file_finder.bEOE THEN
				MoveFile := E_Executer_State.Done;
				_move_file_state := 0;
            ELSE 
                MoveFile := E_Executer_State.Error;
				_move_file_state := 0;
            END_IF
        END_IF
END_CASE
END_METHOD

END_FUNCTION_BLOCK

// ---- POUs/FBs/FB_SQL.TcPOU
FUNCTION_BLOCK FB_SQL
VAR_INPUT
END_VAR
VAR_OUTPUT
END_VAR
VAR
	fbSqlDatabase 			:FB_SQLDatabaseEvt(sNetID := '', tTimeout := T#5S);
	fbSqlCommand 			:FB_SQLCommandEvt(sNetID := '', tTimeout := T#5S);
	fbSqlResult 			:FB_SQLResultEvt(sNetID:='', tTimeout := T#5S); 
	fbSQLStoredProcedure	:FB_SQLStoredProcedureEvt(sNetID:='', tTimeout := T#5S);
	
	nStep					:INT;
	nLastStepError			:INT;
	nConnectionStep			:INT;
	
	// Properties
	_Name					:STRING;
	_DBID					:UINT;
	_RecordCounts			:UDINT;
	_Error					:BOOL;
	_ACK					:BOOL;
	_TimeOut				:TIME := T#5S;
END_VAR

IF _Error THEN
	IF nStep <> 200 THEN
		nLastStepError := nStep;
	END_IF
	nStep := 200;
END_IF
IF _Error AND _ACK THEN
	_Error := FALSE;
	nStep := 0;
END_IF
fbSqlDatabase.tTimeout := _TimeOut;
fbSqlCommand.tTimeout := _TimeOut;
fbSqlResult.tTimeout := _TimeOut;
fbSQLStoredProcedure.tTimeout := _TimeOut;

PROPERTY ACK : BOOL
SET
_ACK := ACK;
END_SET
END_PROPERTY

METHOD PRIVATE Connect : BOOL
VAR_INPUT
END_VAR
Connect := FALSE;
IF fbSqlDatabase.bConnected THEN
	Connect := TRUE;
ELSIF fbSqlDatabase.Connect(_DBID) THEN
	IF fbSqlDatabase.bError THEN
		_Error := TRUE;
		Connect := TRUE;
	ELSE
		Connect := TRUE;
	END_IF
END_IF
END_METHOD

METHOD PRIVATE CreateCmd : BOOL
VAR_INPUT
END_VAR
CreateCmd := FALSE;
IF fbSqlDatabase.CreateCmd(ADR(fbSqlCommand)) THEN
	IF fbSqlDatabase.bError THEN
		_Error := TRUE;
		CreateCmd := TRUE;
	ELSE
		CreateCmd := TRUE;
	END_IF
END_IF
END_METHOD

METHOD PRIVATE CreateSP : BOOL
VAR_INPUT
	sProcedureName		:REFERENCE TO STRING;											//Store Procedure name
    pParameterInfo		:POINTER TO ARRAY [0..MAX_SPPARAMETER] OF ST_SQLSPParameter;	//Parameter Info Array
	nParameterInfoSize	:UDINT;															//Size of parameter info array	
END_VAR
CreateSP := FALSE;
IF fbSQLDatabase.CreateSP(sProcedureName, pParameterInfo, nParameterInfoSize, ADR(fbSQLStoredProcedure)) THEN
	IF fbSQLDatabase.bError THEN
		_Error := TRUE;
		CreateSP := TRUE;
	ELSE
		CreateSP := TRUE;
	END_IF
END_IF
END_METHOD

PROPERTY DBID : UINT
GET
DBID := _DBID;
END_GET
END_PROPERTY

METHOD PRIVATE Disconnect : BOOL
VAR_INPUT
END_VAR
Disconnect := FALSE;
IF fbSqlDatabase.Disconnect() THEN
	IF fbSqlDatabase.bError THEN
		_Error := TRUE;
		Disconnect := TRUE;
	ELSE
		nStep := 0;
		Disconnect := TRUE;
	END_IF
END_IF
END_METHOD

PROPERTY Error : BOOL
GET
Error := _Error;
END_GET
END_PROPERTY

METHOD PRIVATE Execute : BOOL
VAR_INPUT
	sCmd		:REFERENCE TO STRING; 	//SQL command
END_VAR
Execute := FALSE;
IF fbSQLCommand.Execute(ADR(sCmd), SIZEOF(sCmd)) THEN
	IF fbSQLCommand.bError THEN
		_Error := TRUE;
		Execute := TRUE;
	ELSE
		Execute := TRUE;  
	END_IF
END_IF
END_METHOD

METHOD PRIVATE ExecuteDataReturn : BOOL
VAR_INPUT
	sCmd		:REFERENCE TO STRING;	//SQL command
END_VAR
ExecuteDataReturn := FALSE;
IF fbSQLCommand.ExecuteDataReturn(ADR(sCmd), SIZEOF(sCmd), ADR(fbSqlResult)) THEN
	IF fbSQLCommand.bError THEN
		_Error := TRUE;
		ExecuteDataReturn := TRUE;
	ELSE
		ExecuteDataReturn := TRUE;
	END_IF
END_IF
END_METHOD

METHOD ExecuteDataReturnSP : BOOL
VAR_INPUT
	pParameterStrc			:POINTER TO BYTE;												//Parameter struct
	nParameterStrcSize		:UDINT;															//Size of parameter struct
END_VAR
ExecuteDataReturnSP := FALSE;
IF fbSQLStoredProcedure.ExecuteDataReturn(pParameterStrc, nParameterStrcSize, ADR(fbSqlResult)) THEN
	IF fbSQLStoredProcedure.bError THEN
		_Error := TRUE;
		ExecuteDataReturnSP := TRUE;
	ELSE
		ExecuteDataReturnSP := TRUE;
	END_IF    
END_IF
END_METHOD

METHOD Init : BOOL
VAR_INPUT
	sName		:REFERENCE TO STRING;
	nDBID		:REFERENCE TO UINT;
	tTimeout	:REFERENCE TO TIME;
END_VAR
_Name := sName;
_DBID := nDBID;
_TimeOut := tTimeout;
Init := TRUE;
END_METHOD

METHOD Modify : BOOL
VAR_INPUT
	sCmd		:REFERENCE TO STRING; 	//SQL command
END_VAR
Modify := FALSE;
CASE nStep OF 
	0:
		IF Connect() THEN
			nStep := nStep + 20; 
		END_IF
	20:
		IF CreateCmd() THEN
			nStep := nStep + 20;  
		END_IF
		
	40:
		IF Execute(sCmd) THEN
			nStep := nStep + 20; 
		END_IF
	
	60: 
		IF Disconnect() THEN
			nStep := 0;
			Modify := TRUE;
		END_IF
		
	200:
		Modify := TRUE;
END_CASE
END_METHOD

PROPERTY Name : STRING
GET
Name := _Name;
END_GET
END_PROPERTY

METHOD PRIVATE Read : BOOL
VAR_INPUT
	pResultRecord			:POINTER TO BYTE;		//Pointer to the struct
	nResultRecordSize		:REFERENCE TO UDINT;	//Size of the struct
END_VAR
Read := FALSE;
_RecordCounts := fbSQLResult.nDataCount;
IF fbSqlResult.Read(0, _RecordCounts, pResultRecord, nResultRecordSize, TRUE, FALSE) THEN
	IF fbSqlResult.bError THEN
		_Error := TRUE;
		Read := TRUE;
	ELSE
		Read := TRUE;
	END_IF
END_IF
END_METHOD

PROPERTY RecordCounts : UDINT
GET
RecordCounts := _RecordCounts;
END_GET
END_PROPERTY

METHOD PRIVATE ReleaseRead : BOOL
VAR_INPUT
END_VAR
ReleaseRead := FALSE;
IF fbSqlResult.Release() THEN
	IF fbSqlResult.bError THEN
		_Error := TRUE;
		ReleaseRead := TRUE;
	ELSE
		ReleaseRead := TRUE; 
	END_IF
END_IF
END_METHOD

METHOD PRIVATE ReleaseSP : BOOL
VAR_INPUT
END_VAR
ReleaseSP := FALSE;
IF fbSQLStoredProcedure.Release() THEN
	IF fbSQLStoredProcedure.bError THEN
		_Error := TRUE;
		ReleaseSP := TRUE;
	ELSE
		ReleaseSP := TRUE;
	END_IF
END_IF
END_METHOD

METHOD Select : BOOL;
VAR_INPUT
	sCmd					:REFERENCE TO STRING;	//SQL command
	pResultRecord			:POINTER TO BYTE;		//Pointer to the struct
	nResultRecordSize		:UDINT;					//Size of the struct
END_VAR
Select := FALSE;
CASE nStep OF 
	0:
		IF Connect() THEN
			nStep := nStep + 20;  
		END_IF
		
	20:
		IF CreateCmd() THEN
			nStep := nStep + 20;  
		END_IF

	40:
		IF ExecuteDataReturn(sCmd) THEN
			nStep := nStep + 20;
		END_IF
		
	60:
		IF Read(pResultRecord, nResultRecordSize) THEN
			nStep := nStep + 20; 
		END_IF
			
	80: 
		IF ReleaseRead() THEN
			nStep := nStep + 20; 
		END_IF
	
	100:
		IF Disconnect() THEN
			nStep := 0;
			Select := TRUE;
		END_IF
		
	200:
		MEMSET(pResultRecord,0, nResultRecordSize);
		_RecordCounts := 0;
		Select := TRUE;
END_CASE
END_METHOD

METHOD StoredProcedure : BOOL
VAR_INPUT
	sProcedureName		:REFERENCE TO STRING;											//Store Procedure name
    pParameterInfo		:POINTER TO ARRAY [0..MAX_SPPARAMETER] OF ST_SQLSPParameter;	//Parameter Info Array
	nParameterInfoSize	:UDINT;															//Size of parameter info array	
	pParameterStrc		:POINTER TO BYTE;												//Parameter struct
	nParameterStrcSize	:UDINT;															//Size of parameter struct
	pResultRecord		:POINTER TO BYTE;												//Pointer to the struct
	nResultRecordSize	:UDINT;															//Size of the struct
END_VAR
StoredProcedure := FALSE;
CASE nStep OF 
	0:
		IF Connect() THEN
			nStep := nStep + 20;  
		END_IF
		
	20:
		IF CreateSP(sProcedureName, pParameterInfo, nParameterInfoSize) THEN
			nStep := nStep + 20;
		END_IF
		
	40:
		IF ExecuteDataReturnSP(pParameterStrc, nParameterStrcSize) THEN
			nStep := nStep + 20;
		END_IF
		
	60:
		IF Read(pResultRecord, nResultRecordSize) THEN
			nStep := nStep + 20; 
		END_IF
			
	80: 
		IF ReleaseRead() THEN
			nStep := nStep + 20; 
		END_IF
		
	100:
		IF ReleaseSP() THEN
			nStep := nStep + 20; 
		END_IF
	
	120:
		IF Disconnect() THEN
			nStep := 0;
			StoredProcedure := TRUE;
		END_IF
		
	200:
		MEMSET(pResultRecord,0, nResultRecordSize);
		_RecordCounts := 0;
		StoredProcedure := TRUE;
END_CASE
END_METHOD

PROPERTY TimeOut : Time
GET
TimeOut := _TimeOut;
END_GET
END_PROPERTY

END_FUNCTION_BLOCK

// ---- POUs/RobotViseStation/RobotCncProgram.TcPOU
PROGRAM RobotCncProgram
VAR	(* Control *)
	nState						:UDINT;
	nStatePrevious				:UDINT;
	sState						:STRING(500);
	fbCycleTime					:TON;
	nCycleTime					:REAL;
	bError						:	BOOL;
	bInit						:	BOOL := TRUE;
END_VAR
VAR //LastStates
	anLastStates				:ARRAY[0..500] OF UDINT;
    iLastStates					:INT;
END_VAR
VAR (* Robot *)
	fbRobot				: FB_Fanuc;
	arRobotEvents		: ARRAY [0..11] OF TcEventEntry;
END_VAR
VAR	(**)
	
END_VAR
VAR (* Test variables *)
	nOverride			: BYTE := 10;
	bTestEnable			: BOOL;
	nTestIndex			: BYTE;
	nTestCncIndex		: BYTE;
END_VAR
VAR // MySQL
	fbUpdateVise			: FB_SP_spUpdateVise;
	stParameterValues		: ST_ParaVal_UpdateVise;
	fbGetNextVise			: FB_SP_spGetNextVise;
END_VAR
VAR	(*Vise Status handling*)
	i							:	BYTE;
	nUsedViseIndex				:	BYTE;
	nUsedCNC					:	BYTE := 5;
	bActualCNCThreadDone		:	BOOL;
	bActualCNCThreadInBase		:	BOOL;
	bActualCNCProgramNotRunning	:	BOOL;
	nNumberOfEmptyViseSockets	:	BYTE;
	nIndexOfTheEmptySocket		:	BYTE;
END_VAR
VAR (* OPC_UA CNC4*)
	stCNC5_Data					: 	POINTER TO OPC_CNC_Data_Collection;
	tCNC5HeartBeatDelay			: 	TON;
	bCNC5ProgramNotRunning		:	BOOL;
	bCNC5ProgramRunning			:	BOOL;
	bCNC5ServerRunning			:	BOOL;
	bCNC5SystemReady			:	BOOL;
	bCNC5Finished				:	BOOL;
	bCNC5HandshakeTimeout		:	BOOL;
	tCNC5HandshakeTimer			:	TON;
	bCNC5MidwareShutdownPossible	: 	BOOL;	//12500, 14000, cnc4 = 0 or cnc4 >= 50000
	bCNC5ShutdownIsProcessing		:	BOOL;
	
	bOverrideCNC5ProgramUse		:	BOOL := TRUE;
	
	(*CNC 5 Thread State Machine process*)
	nStateCNC5					:	UDINT;
	nStatePreviousCNC5			:	UDINT;
	sStateCNC5					:	STRING(500);
	fbCycleTimeCNC5				:	TON;
	nCycleTimeCNC5				:	REAL;
	bErrorCNC5					:	BOOL;
	bStepEnableCNC5				:	BOOL;
	anLastStatesCNC5			:	ARRAY[0..100] OF UDINT;
    iLastStatesCNC5				:	INT;
	
	//Vise / Term90 / TErm92 / 66.6, 66.7, 67.0 zár-nyit-lefúj
END_VAR
VAR PERSISTENT 
	nRackUsedForCNC4			:	INT;
	nRackUsedForCNC5			:	INT;
	bRobotGoneTowait			:	BOOL;
END_VAR

IF bInit THEN
	FOR i := 1 TO 14 BY 1 DO
		aViseStatus[i].eSocketState := E_ViseSocketState.ViseInSocket;
	END_FOR
	bInit := FALSE;
END_IF


(* =================================== OPC_UA Hearbeat handling =========================================== *)
stCNC5_Data := ADR(OPC_UA_CNC5);
tCNC5HeartBeatDelay(IN := stCNC5_Data^.HeartBeat = 99, PT := T#500MS, Q=>);
IF tCNC5HeartBeatDelay.Q THEN
	stCNC5_Data^.HeartBeat := 0;
END_IF

tCNC5HandshakeTimer(	IN := (stCNC5_Data^.HeartBeat = 0),
						PT := T#3S,
						Q=> bCNC5HandshakeTimeout);
					
(* =================================== OPC_UA Automatic Shutdown handling =========================================== *)					
bCNC5MidwareShutdownPossible := 	nState <= 11000;
								
IF bCNC5MidwareShutdownPossible AND stCNC5_Data^.MidwareRequestedShutdown AND (NOT bCNC5HandshakeTimeout) THEN
	stCNC5_Data^.ApproveShutdownRequest := TRUE;
END_IF

IF stCNC5_Data^.ApproveShutdownRequest THEN
	IF bCNC5HandshakeTimeout THEN
		bCNC5ShutdownIsProcessing := TRUE;
	END_IF
END_IF

IF bCNC5ShutdownIsProcessing THEN
	stCNC5_Data^.ApproveShutdownRequest := FALSE;
	stCNC5_Data^.MidwareRequestedShutdown := FALSE;
	IF (NOT bCNC5HandshakeTimeout) THEN
		bCNC5ShutdownIsProcessing := FALSE;
	END_IF
END_IF
					

(* =================================== Error handling ===================================*)
IF nState > 0 AND nState < 150000 THEN
	nStatePrevious := nState;
END_IF

(* =================================== Maintance =================================== *)
IF bManualModeVise THEN
	nState := 150000;
	nStateCNC5 := 150000;
END_IF


(* =================================== Emergency =================================== *)
IF NOT i_bLO1_CNC45 OR NOT i_bLO2_CNC45 THEN
	nState := 0;
	nStateCNC5 := 0;
END_IF

(* =================================== Last states =================================== *)
IF(nState >= 1000) AND (nState < 150000) THEN
(*Steps before any state*)
	IF anLastStates[0] <> nState THEN
		FOR iLastStates:=500 TO 1 BY -1 DO
			anLastStates[iLastStates]:= anLastStates[iLastStates-1];
		END_FOR
		anLastStates[0]:= nState;
	END_IF
END_IF	

(* =================================== Check common CNC states ===================================*)
bCNC5ProgramNotRunning := stCNC5_Data^.CurentState_Program = 'Idle' OR stCNC5_Data^.CurentState_Program = 'NotSelected' OR stCNC5_Data^.CurentState_Program = 'Interrupted';
bCNC5ProgramRunning := stCNC5_Data^.CurentState_Program = 'Running';
bCNC5ServerRunning := stCNC5_Data^.ServerState = 'Running';
bCNC5SystemReady := stCNC5_Data^.ServerState = 'Running' AND stCNC5_Data^.CurrentState_State = 'NCIsAvailable';
bCNC5Finished := stCNC5_Data^.CurentState_Program = 'Finished';

bStepEnableCNC5 := bStepEnableViseStation;

CASE nUsedCNC OF
	4:
		//Not yet available
	5:
		bActualCNCThreadDone := nStateCNC5 = 50000;
		bActualCNCThreadInBase := nStateCNC5 = 0;
		bActualCNCProgramNotRunning := bCNC5ProgramNotRunning;
END_CASE


(* =================================== Error cases ===================================*)
IF 	fbrobot.bError OR
	stCNC5_Data^.ControlStatus_Error OR
	(NOT bCNC5SystemReady) OR
	(NOT bCNC5ServerRunning) OR 
	(bCNC5HandshakeTimeout AND (NOT bCNC5ShutdownIsProcessing)) OR
	bErrorCNC5
THEN	
	bError := TRUE;
ELSE
	IF bAckP THEN
		bError := FALSE;
	END_IF
END_IF



(* =================================== Cycle time ===================================*)
fbCycleTime(IN:= nState > 11000 AND nState <= 95000, PT:= T#1D, Q=> , ET=> );
IF nState > 10000 AND nState <= 95000 THEN
	nCycleTime := TIME_TO_REAL(fbCycleTime.ET)/1000;
END_IF


MySQL();
CNC5Thread();
Robot();

(*============================================================================================================================================*)
CASE nState OF
	(* Emergency circuit broken - Base state *)
	0:(* Operation stop - Emergency circuit check *)
		sState := CONCAT(UDINT_TO_STRING(nState) ,' - A biztonsági kör nem aktív');
		
		fbRobot.eCommand := E_Robot_Command.NoCommand;
		fbRobot.nViseNumber := 0;
		fbRobot.nCncNumber := 0;
		
		stCNC5_Data^.DoorControl_CloseDoor := FALSE;
		stCNC5_Data^.DoorControl_OpenDoor := FALSE;
		stCNC5_Data^.MagazineTable_Trigger := FALSE;
		stCNC5_Data^.ToolTable_Trigger := FALSE;
		stCNC5_Data^.M401_Acknowledge := FALSE;
		stCNC5_Data^.M402_Acknowledge := FALSE;
		stCNC5_Data^.M403_Acknowledge := FALSE;
		stCNC5_Data^.StartCNCProgram := FALSE;
		stCNC5_Data^.StopCNCProgram := FALSE;
		stCNC5_Data^.CancelCNCProgram := FALSE;
		stCNC5_Data^.SelectCNCProgramByNodeID := FALSE;
		stCNC5_Data^.SelectCNCPrograBlockNumber := FALSE;
		stCNC5_Data^.ToolTableLoadTrigger := FALSE;
		stCNC5_Data^.MagazineTableLoadTrigger := FALSE;
		stCNC5_Data^.ProgramLoadTrigger := FALSE;
		
		GVL_IO.q_bCNC4_Fix_Vise := TRUE;
		GVL_IO.q_bCNC4_Release_Vise := FALSE;
		bRobotGoneTowait := FALSE;
		
		IF i_bLO1_CNC45 AND i_bLO2_CNC45 AND (NOT bManualModeVise) AND (NOT bError) THEN
			IF bStepEnableViseStation THEN
				nState := nState + 20;
			END_IF
		END_IF

	20: 
		sState := CONCAT(UDINT_TO_STRING(nState) ,' - Robot alaphelyzetfelvétel');
		fbRobot.eCommand := E_Robot_Command.Home;
		IF NOT fbRobot.bBusy AND fbRobot.bReady THEN
			IF bStepEnableViseStation THEN
				fbRobot.eCommand := E_Robot_Command.NoCommand;
				nState := nState + 20;
			END_IF
		END_IF

	40:
		nState := 100;
		
	100:		(*-----=== CNC ellenőrzés ===-----*)
		sState := CONCAT(UDINT_TO_STRING(nState) ,' - A CNC 5 ellenőrzése');
		IF stCNC5_Data^.ServerState = 'Running' AND
		   stCNC5_Data^.CurrentState_State = 'NCIsAvailable' THEN
				IF stCNC5_Data^.CurentState_Program = 'Running' THEN
					IF bStepEnableViseStation THEN
						nState := 11700;										// A megmunkálás folyamatban -> Várakozás megmunkálás végére.
					END_IF
				ELSIF	stCNC5_Data^.CurentState_Program = 'Idle' OR stCNC5_Data^.CurentState_Program = 'NotSelected' OR stCNC5_Data^.CurentState_Program = 'Interrupted' THEN
					IF stDutData_Cnc1.nDutId > 0 AND stDutData_Cnc1.bDone THEN 
						IF bStepEnableViseStation THEN									// Késztermék a satuban
							nState := 120;
						END_IF
					ELSE
						IF bStepEnableViseStation THEN									// A satu üres
							nState := 120;
						END_IF
					END_IF
				END_IF
		END_IF

	120:		(*-----=== CNC ajtó nnyitása ===-----*)
		sState := CONCAT(UDINT_TO_STRING(nState) ,' - A 5.CNC ajtó nyitása');
		
		stCNC5_Data^.DoorControl_OpenDoor := TRUE;
		IF stCNC5_Data^.DoorControl_DoorOpened THEN
			IF bStepEnableViseStation THEN	
				stCNC5_Data^.DoorControl_OpenDoor := FALSE;
				nState := 500;
			END_IF
		END_IF
		
	500:
		IF bStepEnableViseStation THEN
			nState := 11000;
		END_IF

	(*Check for next possible process *)	
	11000:
		sState := CONCAT(UDINT_TO_STRING(nState) ,' - Következő folyamatra várakozás');
	
		(*Currently (2023.11.09) Only CNC 5 is available. This way, CNC is constantly 5 yet*)
		nUsedCNC := 5;
		
		IF fbRobot.RobotIn.Status.bVisePresent THEN
			nState  := 11500;
		ELSIF stCNC5_Data^.ApproveShutdownRequest THEN
			nState  := 11010;
		(*Check if there is a Ready to CNC Vise *)
		ELSIF (CheckForViseStatus(E_Vise_State.ReadyToCnc) >= ViseProgram.nStartIndex) AND (CheckForViseStatus(E_Vise_State.ReadyToCnc) <= ViseProgram.nMaxIndex) AND (CheckForViseStatus(E_Vise_State.CncDone) = 99) AND (CheckForViseStatus(E_Vise_State.ReadyToCnc) <> 99) AND (bActualCNCProgramNotRunning AND (bActualCNCThreadInBase)) THEN
			
			nUsedViseIndex := CheckForViseStatus(E_Vise_State.ReadyToCnc);
			
			CASE nUsedCNC OF
				4: nRackUsedForCNC4 := nUsedViseIndex;
				5: nRackUsedForCNC5 := nUsedViseIndex;
				ELSE ; (*Else is not relevant in this case, because of the pre-condition*)
			END_CASE
		
			IF bActualCNCProgramNotRunning AND (bActualCNCThreadInBase) THEN
				IF (CheckForViseStatus(E_Vise_State.InCnc) = 99) AND (CheckForViseStatus(E_Vise_State.CncDone) = 99) (*AND (CheckForUsedCNCByVise(nUsedCNC) <> nUsedCNC)*) THEN	//No vise with CncDone and InCNC Status in the requested CNC
					IF CheckAllViseInSafePos() THEN
						IF (NOT fbRobot.bBusy) THEN
							bRobotGoneTowait := FALSE;
							nState := 12000;	//Pick vise from socket, put into CNC
						END_IF
					END_IF
				END_IF
			END_IF
		
			
		ELSIF (CheckForViseStatus(E_Vise_State.CncDone) >= ViseProgram.nStartIndex) AND (CheckForViseStatus(E_Vise_State.CncDone) <= ViseProgram.nMaxIndex) AND (CheckForViseStatus(E_Vise_State.CncDone) <> 99) THEN
			
			nUsedViseIndex := CheckForViseStatus(E_Vise_State.CncDone);
		
			CASE nUsedCNC OF
				4: nRackUsedForCNC4 := nUsedViseIndex;
				5: nRackUsedForCNC5 := nUsedViseIndex;
				ELSE ; (*Else is not relevant in this case, because of the pre-condition*)
			END_CASE

			IF (bActualCNCThreadDone) THEN
				IF CheckAllViseInSafePos() THEN
					IF (NOT fbRobot.bBusy) THEN
						bRobotGoneTowait := FALSE;
						nState := 14000;	//Pick vise from CNC, Put it to its socket
					END_IF
				END_IF
			END_IF
		//If none of the above ran, then send the robot to Wait pos (Prg2)
		ELSIF (NOT fbRobot.bBusy) AND (NOT bRobotGoneTowait) THEN
			nState := 16000;
		END_IF
		
	(*Wait for CNC to finish shutdown*)		
	11010:
		sState := CONCAT(UDINT_TO_STRING(nState) ,' - Waiting for OPC midware to restart');
	 	IF (NOT bCNC5HandshakeTimeout) AND (NOT bCNC5ShutdownIsProcessing) THEN
			nState := 11000;
		END_IF
	
	11500:
		sState := CONCAT(UDINT_TO_STRING(nState) ,' - Robot megfogóban satu van. Üres satu foglalatok ellenőrzése');	
		
		FOR i := ViseProgram.nStartIndex TO ViseProgram.nMaxIndex BY 1 DO 
			IF aViseStatus[i].eSocketState = E_ViseSocketState.SocketEmpty THEN
				nNumberOfEmptyViseSockets := nNumberOfEmptyViseSockets + 1;
			END_IF
		END_FOR
		nState  := nState + 20;
		
	11520:
		IF nNumberOfEmptyViseSockets = 1 THEN
			FOR i := ViseProgram.nStartIndex TO ViseProgram.nMaxIndex BY 1 DO 
				IF aViseStatus[i].eSocketState = E_ViseSocketState.SocketEmpty THEN
					sState := CONCAT(UDINT_TO_STRING(nState) , CONCAT(' - Üres satu foglalat található a ' , CONCAT( BYTE_TO_STRING(i),' indexű helyen')));	
					nIndexOfTheEmptySocket := i;
					EXIT;
				END_IF
			END_FOR
		ELSIF nNumberOfEmptyViseSockets = 0 THEN
			sState := CONCAT(UDINT_TO_STRING(nState) ,' - Nem található üres satu foglalat. Rakassa le a robottal a satut.');
			nState := 11521;	
		ELSE
			sState := CONCAT(UDINT_TO_STRING(nState) ,' - Több üres foglalat található. Rakassa le a robottal a satut.');
		END_IF 
		
		nState := nState + 20;
		
	11540:
		//Innen egyelőre kézzel lép tovább
		
	11560:
		sState := CONCAT(UDINT_TO_STRING(nState) , CONCAT(' - Robot satu visszarakás erre a satu foglalatra ', BYTE_TO_STRING(nIndexOfTheEmptySocket)));
		
		fbRobot.nViseNumber := nUsedViseIndex;
		fbRobot.nCncNumber := nUsedCNC;
		fbRobot.eCommand := E_Robot_Command.Put_Down_Vise;
		
		IF fbRobot.bBusy THEN
			nState := 11580;
		END_IF
		
	11580:
		sState := CONCAT(UDINT_TO_STRING(nState) ,' - Várakozás robot satu visszarakásra');
		
		IF (NOT fbRobot.bBusy) THEN
			nState := 11600;
		END_IF
		
	11600:
		nState := 11000;
		
	11700:
		sState := CONCAT(UDINT_TO_STRING(nState) ,' - CNC program befejezésre várakozás');	
		
		
	(*Pick vise from requested rack, and place it into the requested CNC*)
	12000:
		sState := CONCAT(UDINT_TO_STRING(nState) ,' - Robot alaphelyzetfelvétel');
		
		fbRobot.eCommand := E_Robot_Command.Home;
		
		IF fbRobot.bBusy THEN
			nState := 12005;
		END_IF
		
	12005:
		sState := CONCAT(UDINT_TO_STRING(nState) ,' - Robot alaphelyzetre mozgásra vár');
		
		IF (NOT fbRobot.bBusy) THEN
			fbRobot.eCommand := E_Robot_Command.NoCommand;
			IF bStepEnableViseStation THEN
				nState := 12010;
			END_IF
		END_IF
		
	12010:
		sState := CONCAT(UDINT_TO_STRING(nState) ,' - Kért satu henger munkahelyzetre');
		
		fbViseStation[nUsedViseIndex].Vise.bBasePosCmd := FALSE;
		fbViseStation[nUsedViseIndex].Vise.bWorkPosCmd := TRUE;
		
		IF fbViseStation[nUsedViseIndex].Vise.bWorkPosStab OR bAckP THEN
			IF bStepEnableViseStation THEN
				nState := nState + 10;
			END_IF
		END_IF
		
	12020:
		sState := CONCAT(UDINT_TO_STRING(nState) ,' - Robot betöltő állomásról satu felvételre indul');
		
		fbRobot.nViseNumber := nUsedViseIndex;
		fbRobot.nCncNumber := nUsedCNC;
		fbRobot.eCommand := E_Robot_Command.Pick_Up_Vise;
		
		IF fbRobot.bBusy THEN
			nState := 12080;
		END_IF
		
	12080:
		sState := CONCAT(UDINT_TO_STRING(nState) ,' - Várakozás robotprogram végére');
		
		IF (NOT fbRobot.bBusy) THEN
			IF bStepEnableViseStation THEN
				fbViseStation[nUsedViseIndex].Vise.bWorkPosCmd := FALSE;
				aViseStatus[nUsedViseIndex].eState := E_Vise_State.InRobotArmBeforeCnc;
				aViseStatus[nUsedViseIndex].eSocketState := E_ViseSocketState.SocketEmpty;
				fbRobot.eCommand := E_Robot_Command.NoCommand;
				nState := 12100;
			END_IF
		END_IF
		
	12100:
		sState := CONCAT(UDINT_TO_STRING(nState) ,' - Kért satu henger alaphelyzetre');
		
		fbViseStation[nUsedViseIndex].Vise.bBasePosCmd := TRUE;
		fbViseStation[nUsedViseIndex].Vise.bWorkPosCmd := FALSE;
		
		IF fbViseStation[nUsedViseIndex].Vise.bBasePosStab THEN
			IF bStepEnableViseStation THEN
				nState := 12500;
			END_IF
		END_IF
		
		
	12500:	
		sState := CONCAT(UDINT_TO_STRING(nState) ,' - CNC ajtó nyitott állapot ellenőrzés , Satu fixer elenged');
		
		CASE nUsedCNC OF
			4:
				//Not yet available
			5:
				GVL_IO.q_bCNC4_Fix_Vise := FALSE;
				GVL_IO.q_bCNC4_Release_Vise := TRUE;
				IF CheckAndOpenCNCDoor(5) THEN
					IF bStepEnableViseStation THEN
						nState := nState + 20;
					END_IF
				END_IF
		END_CASE
		
	12520:
		sState := CONCAT(UDINT_TO_STRING(nState) ,' - Robot CNC-be satu berakásra indul');
		
		fbRobot.nViseNumber := nUsedViseIndex;
		fbRobot.nCncNumber := nUsedCNC;
		fbRobot.eCommand := E_Robot_Command.Put_Down_Cnc;
		
		IF fbRobot.bBusy THEN
			nState := 12580;
		END_IF
		
	12580:
		sState := CONCAT(UDINT_TO_STRING(nState) ,' - Várakozás robotprogram végére, Satu fixer rögzít');
		
		IF (NOT fbRobot.bBusy) THEN
			
			aViseStatus[nUsedViseIndex].eState := E_Vise_State.InCnc;
			aViseStatus[nUsedViseIndex].nInCNC := nUsedCNC;
			fbRobot.eCommand := E_Robot_Command.NoCommand;
			
			CASE nUsedCNC OF
				4:
					//Not yet available
				5:
					GVL_IO.q_bCNC4_Fix_Vise := TRUE;
					GVL_IO.q_bCNC4_Release_Vise := FALSE;	
			END_CASE
			
			IF bStepEnableViseStation THEN
				nState := nState + 20;
			END_IF
		END_IF
		
	12600:
		sState := CONCAT(UDINT_TO_STRING(nState) ,' - Robot WAIT pozícióra indul');
		
		fbRobot.nViseNumber := nUsedViseIndex;
		fbRobot.nCncNumber := nUsedCNC;
		fbRobot.eCommand := E_Robot_Command.Wait;
		
		IF fbRobot.bBusy THEN
			nState := nState + 20;
		END_IF
		
	12620:
		sState := CONCAT(UDINT_TO_STRING(nState) ,' - Robot WAIT pozícióra várakozás');
	
		IF (NOT fbRobot.bBusy) THEN
			
			fbRobot.eCommand := E_Robot_Command.NoCommand;
			
			IF bStepEnableViseStation THEN
				IF (TRUE) THEN
					nState := nState + 20;
				ELSE
					nState := 13000;
				END_IF
			END_IF
		END_IF
		
	12640:
		sState := CONCAT(UDINT_TO_STRING(nState) ,' - CNC állapotgép indítása');
		
		CASE nUsedCNC OF
			4:
				//Not yet available
			5:
				IF (NOT bErrorCNC5) THEN
					IF bStepEnableViseStation THEN
						nStateCNC5 := 1000;
						nState := nState + 20;
					END_IF
				END_IF
		END_CASE
		
		
	12660:
		sState := CONCAT(UDINT_TO_STRING(nState) ,' - CNC állapotgép indulás ellenőrzés');
		
		CASE nUsedCNC OF
			4:
				//Not yet available				
			5:
				IF (NOT bErrorCNC5) THEN
					IF nStateCNC5 > 1000 THEN
						nState := 13000;
					END_IF
				END_IF
		END_CASE
		
		
	13000:
		sState := CONCAT(UDINT_TO_STRING(nState) ,' - CNC állapotgép elindult. Vissza várakozó helyzetbe!');
		(*CNC Started. Go to base pos, check if put-in needed, or finished.*)
		IF bStepEnableViseStation THEN
			nState := 11000;
		END_IF
	
	
		
	
	
	(*Pick vise from requested CNC, and place it into the requested rack*)
	14000:
		sState := CONCAT(UDINT_TO_STRING(nState) ,' - Robot alaphelyzetfelvétel');
		
		fbRobot.eCommand := E_Robot_Command.Home;
		
		IF fbRobot.bBusy THEN
			nState := 14005;
		END_IF
		
	14005:
		sState := CONCAT(UDINT_TO_STRING(nState) ,' - Robot alaphelyzetre mozgásra vár');
		
		IF (NOT fbRobot.bBusy) THEN
			fbRobot.eCommand := E_Robot_Command.NoCommand;
			IF bStepEnableViseStation THEN
				nState := 14010;
			END_IF
		END_IF
		
	14010:	
		sState := CONCAT(UDINT_TO_STRING(nState) ,' - CNC ajtó nyitott állapot ellenőrzés , Satu fixer elenged');
		
		CASE nUsedCNC OF
			4:
				//Not yet available
			5:
				nStateCNC5 := 0;
				GVL_IO.q_bCNC4_Fix_Vise := FALSE;
				GVL_IO.q_bCNC4_Release_Vise := TRUE;
				IF CheckAndOpenCNCDoor(5) THEN
					IF bStepEnableViseStation THEN
						nState := nState + 10;
					END_IF
				END_IF
		END_CASE
		
	14020:
		sState := CONCAT(UDINT_TO_STRING(nState) ,' - Robot CNC-ből satu kivétel indul');
		
		fbRobot.nViseNumber := nUsedViseIndex;
		fbRobot.nCncNumber := nUsedCNC;
		fbRobot.eCommand := E_Robot_Command.Pick_Up_Cnc;
		
		IF fbRobot.bBusy THEN
			nState := 14080;
		END_IF
		
	14080:
		sState := CONCAT(UDINT_TO_STRING(nState) ,' - Várakozás robotprogram végére, Satu fixer rögzít');
		
		IF (NOT fbRobot.bBusy) THEN
			
			aViseStatus[nUsedViseIndex].eState := E_Vise_State.InRobotArmAfterCnc;
			aViseStatus[nUsedViseIndex].nInCNC := 0;
			fbRobot.eCommand := E_Robot_Command.NoCommand;
			
			CASE nUsedCNC OF
				4:
					//Not yet available					
				5:
					GVL_IO.q_bCNC4_Fix_Vise := TRUE;
					GVL_IO.q_bCNC4_Release_Vise := FALSE;
					IF bStepEnableViseStation THEN
						nState := 14500;
					END_IF
			END_CASE
		END_IF
		
	14500:
		sState := CONCAT(UDINT_TO_STRING(nState) ,' - Kért satu henger munkahelyzetre');
		
		fbViseStation[nUsedViseIndex].Vise.bBasePosCmd := FALSE;
		fbViseStation[nUsedViseIndex].Vise.bWorkPosCmd := TRUE;
		
		IF fbViseStation[nUsedViseIndex].Vise.bWorkPosStab OR bAckP THEN
			IF bStepEnableViseStation THEN
				nState := nState + 20;
			END_IF
		END_IF
		
	14520:
		sState := CONCAT(UDINT_TO_STRING(nState) ,' - Robot CNCből satu kivétel után betöltő állomásra indul');
		
		fbRobot.nViseNumber := nUsedViseIndex;
		fbRobot.nCncNumber := nUsedCNC;
		fbRobot.eCommand := E_Robot_Command.Put_Down_Vise;
		
		IF fbRobot.bBusy THEN
			nState := 14580;
		END_IF
		
	14580:
		sState := CONCAT(UDINT_TO_STRING(nState) ,' - Várakozás robotprogram végére');
		
		IF (NOT fbRobot.bBusy) THEN
			
			fbViseStation[nUsedViseIndex].Vise.bWorkPosCmd := FALSE;
			aViseStatus[nUsedViseIndex].eState := E_Vise_State.OutForUnload;
			aViseStatus[nUsedViseIndex].eSocketState := E_ViseSocketState.ViseInSocket;
			fbRobot.eCommand := E_Robot_Command.NoCommand;
			
			IF bStepEnableViseStation THEN
				nState := 14600;
			END_IF
		END_IF
		
	14600:
		sState := CONCAT(UDINT_TO_STRING(nState) ,' - Kért satu henger alaphelyzetre');
		
		fbViseStation[nUsedViseIndex].Vise.bBasePosCmd := TRUE;
		fbViseStation[nUsedViseIndex].Vise.bWorkPosCmd := FALSE;
		
		IF fbViseStation[nUsedViseIndex].Vise.bBasePosStab THEN
			IF bStepEnableViseStation THEN
				nState := 15000;
			END_IF
		END_IF
		
		
	15000:
		sState := CONCAT(UDINT_TO_STRING(nState) ,' - Satu előkészítő állomásra visszarakás kész');	
		
		IF bStepEnableViseStation THEN
			nState := 11000;
		END_IF
		
		
	(*No process requested. Send the robot to park*)
	16000:
		sState := CONCAT(UDINT_TO_STRING(nState) ,' - Várakozás hogy robot ne legyen Busy');	
		
		IF (NOT fbRobot.bBusy) THEN
			IF bStepEnableViseStation THEN
				nState := nState + 20;
			END_IF
		END_IF
		
	16020:
		sState := CONCAT(UDINT_TO_STRING(nState) ,' - Robot WAIT pozícióra indul');
		
		fbRobot.eCommand := E_Robot_Command.Wait;
		
		IF fbRobot.bBusy THEN
			nState := nState + 20;
		END_IF
		
	16040:
		sState := CONCAT(UDINT_TO_STRING(nState) ,' - Robot WAIT pozícióra várakozás');
	
		IF (NOT fbRobot.bBusy) THEN
			
			fbRobot.eCommand := E_Robot_Command.NoCommand;
			bRobotGoneTowait := TRUE;
			
			IF bStepEnableViseStation THEN
				nState := 11000;
			END_IF
		END_IF
	
	150000: (* Maintenance *)
		sState := CONCAT(UDINT_TO_STRING(nState) ,' - Maintenance');
		IF NOT bManualModeVise THEN
			nState := 0;
		END_IF
		
	200000:(* Error handling *)
		sState := CONCAT(UDINT_TO_STRING(nState) ,CONCAT(' - Error, from this state: ' , sState));
		nState := 200020;

	200020:(* Error handling *)
		IF bAckP THEN
			CASE nStatePrevious OF
				0..9999: nState := 0;
				10000..25000: nState := 10000;
				30000..31000: nState := 30000;
			ELSE nState := 0;
			END_CASE
		END_IF	
		
	ELSE //Not a real step, for test purposes
		sState := CONCAT(UDINT_TO_STRING(nState) ,' - Not a real step, for test purposes');
END_CASE

METHOD INTERNAL CheckAllViseInSafePos : BOOL
VAR
	i	:	INT;
END_VAR
(*Check if all Vises ar in base position*)

FOR i := ViseProgram.nStartIndex TO ViseProgram.nMaxIndex BY 1 DO
	IF (NOT fbViseStation[i].Vise.bBasePosStab) AND (aViseStatus[1].eState <> E_Vise_State.OutOfService) THEN
		CheckAllViseInSafePos := FALSE;
		RETURN;
	END_IF
END_FOR

CheckAllViseInSafePos := TRUE;
RETURN;
END_METHOD

METHOD INTERNAL CheckAndOpenCNCDoor : BOOL
VAR_INPUT
	nActualCNC	:	BYTE;
END_VAR

CASE nActualCNC OF
	4:
		//Not yet available
	5:
		IF stCNC5_Data^.DoorControl_DoorOpened THEN
			CheckAndOpenCNCDoor := TRUE;
			RETURN;
		ELSE
			stCNC5_Data^.DoorControl_OpenDoor := TRUE;
			IF stCNC5_Data^.DoorControl_DoorOpened THEN
				IF bStepEnable THEN	
					stCNC5_Data^.DoorControl_OpenDoor := FALSE;
					CheckAndOpenCNCDoor := TRUE;
					RETURN;
				END_IF
			END_IF
		END_IF
		
END_CASE
END_METHOD

METHOD INTERNAL CheckForUsedCNCByVise : BYTE
VAR_INPUT
	nCncUsed		:	BYTE;
END_VAR
VAR
	i					:	BYTE;
END_VAR
FOR i := ViseProgram.nStartIndex TO ViseProgram.nMaxIndex BY 1 DO
	IF aViseStatus[i].nInCNC = nCncUsed THEN
		CheckForUsedCNCByVise := i;
		RETURN;
	END_IF
END_FOR
CheckForUsedCNCByVise := 99;
RETURN;
END_METHOD

METHOD INTERNAL CheckForViseStatus : BYTE
VAR_INPUT
	i_stViseState		:	E_Vise_State;
END_VAR
VAR
	i					:	BYTE;
END_VAR

FOR i := ViseProgram.nStartIndex TO ViseProgram.nMaxIndex BY 1 DO
	IF aViseStatus[i].eState = i_stViseState THEN
		CheckForViseStatus := i;
		RETURN;
	END_IF
END_FOR
CheckForViseStatus := 99;
RETURN;
END_METHOD

ACTION CNC5Thread:
	
(* =================================== Error handling ===================================*)
IF nStateCNC5 > 0 AND nStateCNC5 < 150000 THEN
	nStatePreviousCNC5 := nStateCNC5;
END_IF

(* =================================== Last states =================================== *)
IF(nStateCNC5 >= 1000) AND (nStateCNC5 < 150000) THEN
(*Steps before any state*)
	IF anLastStatesCNC5[0] <> nStateCNC5 THEN
		FOR iLastStatesCNC5 := 100 TO 1 BY -1 DO
			anLastStatesCNC5[iLastStatesCNC5]:= anLastStatesCNC5[iLastStatesCNC5-1];
		END_FOR
		anLastStatesCNC5[0]:= nStateCNC5;
	END_IF
END_IF	

	
CASE nStateCNC5 OF
				(*-----=== Alaphelyzet, startra várakozás ===-----*)
	0:
		sStateCNC5 := CONCAT(UDINT_TO_STRING(nStateCNC5) ,' - Idle');
		
	1000:
		nStateCNC5 := 13000;
	
	13000:		(*-----=== CNC ajtó zárása ===-----*)
		sStateCNC5 := CONCAT(UDINT_TO_STRING(nStateCNC5) ,' - A CNC ajtó zárása');
		stCNC5_Data^.DoorControl_CloseDoor := TRUE;
		IF stCNC5_Data^.DoorControl_DoorClosed THEN
			IF bStepEnableCNC5 THEN	
				stCNC5_Data^.DoorControl_CloseDoor := FALSE;
				nStateCNC5 := nStateCNC5 + 20;
			END_IF
		END_IF

	13020:		(*-----=== CNC előkészítése ===-----*)
		sStateCNC5 := CONCAT(UDINT_TO_STRING(nStateCNC5) ,' - A CNC előkészítése');
		IF TRUE THEN															// Külön FB-be rakni mert még képlékeny CAM file letöltése, ellenőrzése, felmásolása, betöltése, ........ 
			IF bStepEnableCNC5 THEN	
				nStateCNC5 := nStateCNC5 + 20;
			END_IF
		END_IF

	13040:		(*-----=== CAM program indítása ===-----*)
		sStateCNC5 := CONCAT(UDINT_TO_STRING(nStateCNC5) ,' - CAM program indítása');
		stCNC5_Data^.StartCNCProgram := TRUE;
		IF stCNC5_Data^.CurentState_Program = 'Running' THEN
			IF bStepEnableCNC5 THEN	
				stCNC5_Data^.StartCNCProgram := FALSE;
				nStateCNC5 := 13100;
			END_IF
		END_IF
		
	13100:		(*-----=== Várakozás CAM program végére ===-----*)
		sStateCNC5 := CONCAT(UDINT_TO_STRING(nStateCNC5) ,' - Várakozás CAM program végére');
		IF stCNC5_Data^.CurentState_Program = 'Finished' OR stCNC5_Data^.CurentState_Program = 'Idle' THEN
			IF bStepEnableCNC5 THEN	
				aViseStatus[nRackUsedForCNC5].eState := E_Vise_State.CncDone;
				stCNC5_Data^.DoorControl_CloseDoor := FALSE;
				nStateCNC5 := nStateCNC5 + 20;
			END_IF
		END_IF

	13120:		(*-----=== CNC folyamat befejezése ===-----*)
		sStateCNC5 := CONCAT(UDINT_TO_STRING(nStateCNC5) ,' - A CNC folyamat befejezése');
		IF TRUE THEN															// Külön FB-be rakni mert még képlékeny: minőségellenőrzés, mérési adatok, .... 
			IF bStepEnableCNC5 THEN	
				nStateCNC5 := nStateCNC5 + 20;
			END_IF
		END_IF

	13140:		(*-----=== CAM program leállítása ===-----*)
		sStateCNC5 := CONCAT(UDINT_TO_STRING(nStateCNC5) ,' - CAM program leállítása');
		stCNC5_Data^.CancelCNCProgram := TRUE;
		IF stCNC5_Data^.CurentState_Program = 'Idle' THEN
			IF bStepEnableCNC5 THEN	
				stCNC5_Data^.CancelCNCProgram := FALSE;
				nStateCNC5 := nStateCNC5 + 20;
			END_IF
		END_IF

	13160:		(*-----=== CNC ajtó nnyitása ===-----*)
		sStateCNC5 := CONCAT(UDINT_TO_STRING(nStateCNC5) ,' - A CNC ajtó nyitása');
		stCNC5_Data^.DoorControl_OpenDoor := TRUE;
		IF stCNC5_Data^.DoorControl_DoorOpened THEN
			IF bStepEnableCNC5 THEN	
				stCNC5_Data^.DoorControl_OpenDoor := FALSE;
				nStateCNC5 := 50000;
			END_IF
		END_IF
		
		
	50000:
		sStateCNC5 := CONCAT(UDINT_TO_STRING(nStateCNC5) ,' - Szülő program nyugtájára várakozás');
		
		
		
	150000: (* Maintenance *)
		sStateCNC5 := CONCAT(UDINT_TO_STRING(nStateCNC5) ,' - Maintenance');
		IF NOT bManualModeVise THEN
			nStateCNC5 := 0;
		END_IF
		
		
	200000:(* Error handling *)
		sStateCNC5 := CONCAT(UDINT_TO_STRING(nStateCNC5) ,CONCAT(' - Error, from this state: ' , sStateCNC5));
		nStateCNC5 := 200020;

	200020:(* Error handling *)
		IF bAckP THEN
			CASE nStatePreviousCNC5 OF
				0..149999: nStateCNC5 := 0;
			ELSE nStateCNC5 := 0;
			END_CASE
		END_IF	
		
	ELSE //Not a real step, for test purposes
		sStateCNC5 := CONCAT(UDINT_TO_STRING(nStateCNC5) ,' - Not a real step, for test purposes');
		
		
END_CASE
END_ACTION

ACTION MySQL:
fbGetNextVise(
	Target:= , 
	nRecordStartIndex:= , 
	tTimeout:= , 
	bExecute:= , 
	bBusy=> , 
	bError=> , 
	ipResult=> , 
	nViseNr=> );

fbUpdateVise(
	nRecordStartIndex:= , 
	tTimeout:= , 
	bExecute:= , 
	bBusy=> , 
	bError=> , 
	ipResult=> , 
	stParameterValues:= stParameterValues);
END_ACTION

ACTION Robot:
arRobotEvents[0] := TC_EVENTS.MyEvents.RobotNoPneumaticsErr;
arRobotEvents[1] := TC_EVENTS.MyEvents.RobotNotCorrectPrgErr;
arRobotEvents[2] := TC_EVENTS.MyEvents.RobotNotProdOnRobotErr;
arRobotEvents[3] := TC_EVENTS.MyEvents.RobotProdOnRobotErr;
arRobotEvents[4] := TC_EVENTS.MyEvents.RobotGripperOpenErr;
arRobotEvents[5] := TC_EVENTS.MyEvents.RobotGripperCloseErr;
arRobotEvents[6] := TC_EVENTS.MyEvents.RobotNotCorrectViseNumberErr;
arRobotEvents[7] := TC_EVENTS.MyEvents.RobotNotReadyErr;
arRobotEvents[8] := TC_EVENTS.MyEvents.RobotBasePosErr;

(*-----=== Hand shake jelek kezelése ===-----*)
fbRobot.bVise_1_7_Reset := 		fbRobot.bVise_1_7_Set AND_THEN CheckAllViseInSafePos();

fbRobot.bVise_8_14_Reset := 	fbRobot.bVise_8_14_Set AND_THEN CheckAllViseInSafePos();

